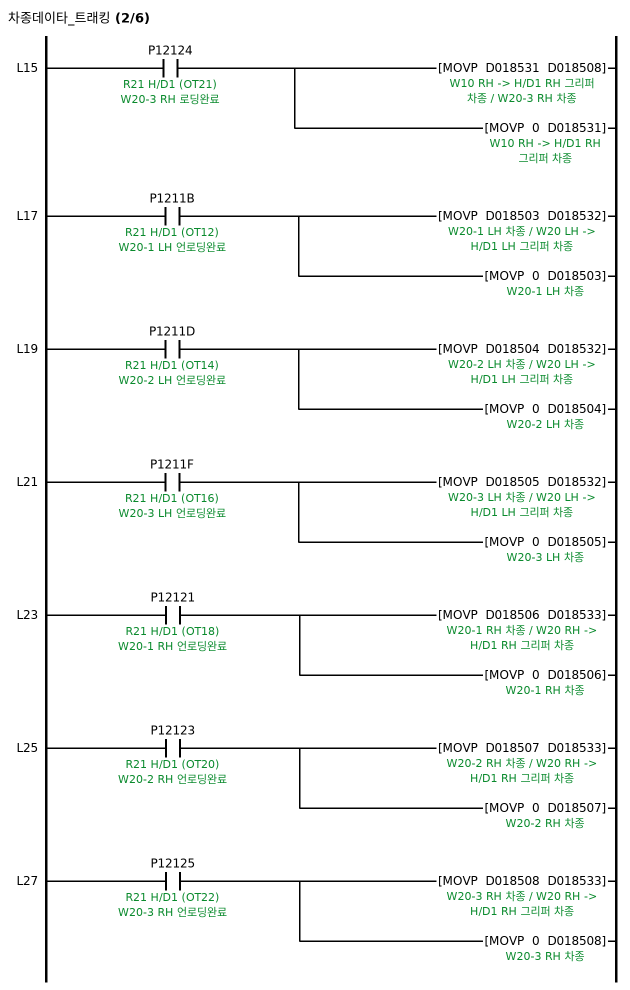
[picture p432: 차종데이타_트래킹 rungs L15-L27]
; L15
LOAD      P12124	// R21 H/D1 (OT21) W20-3 RH 로딩완료
MOVP      D018531 D018508	// W10 RH -> H/D1 RH 그리퍼 차종 / W20-3 RH 차종
MOVP      0 D018531	// W10 RH -> H/D1 RH 그리퍼 차종
; L17
LOAD      P1211B	// R21 H/D1 (OT12) W20-1 LH 언로딩완료
MOVP      D018503 D018532	// W20-1 LH 차종 / W20 LH -> H/D1 LH 그리퍼 차종
MOVP      0 D018503	// W20-1 LH 차종
; L19
LOAD      P1211D	// R21 H/D1 (OT14) W20-2 LH 언로딩완료
MOVP      D018504 D018532	// W20-2 LH 차종 / W20 LH -> H/D1 LH 그리퍼 차종
MOVP      0 D018504	// W20-2 LH 차종
; L21
LOAD      P1211F	// R21 H/D1 (OT16) W20-3 LH 언로딩완료
MOVP      D018505 D018532	// W20-3 LH 차종 / W20 LH -> H/D1 LH 그리퍼 차종
MOVP      0 D018505	// W20-3 LH 차종
; L23
LOAD      P12121	// R21 H/D1 (OT18) W20-1 RH 언로딩완료
MOVP      D018506 D018533	// W20-1 RH 차종 / W20 RH -> H/D1 RH 그리퍼 차종
MOVP      0 D018506	// W20-1 RH 차종
; L25
LOAD      P12123	// R21 H/D1 (OT20) W20-2 RH 언로딩완료
MOVP      D018507 D018533	// W20-2 RH 차종 / W20 RH -> H/D1 RH 그리퍼 차종
MOVP      0 D018507	// W20-2 RH 차종
; L27
LOAD      P12125	// R21 H/D1 (OT22) W20-3 RH 언로딩완료
MOVP      D018508 D018533	// W20-3 RH 차종 / W20 RH -> H/D1 RH 그리퍼 차종
MOVP      0 D018508	// W20-3 RH 차종

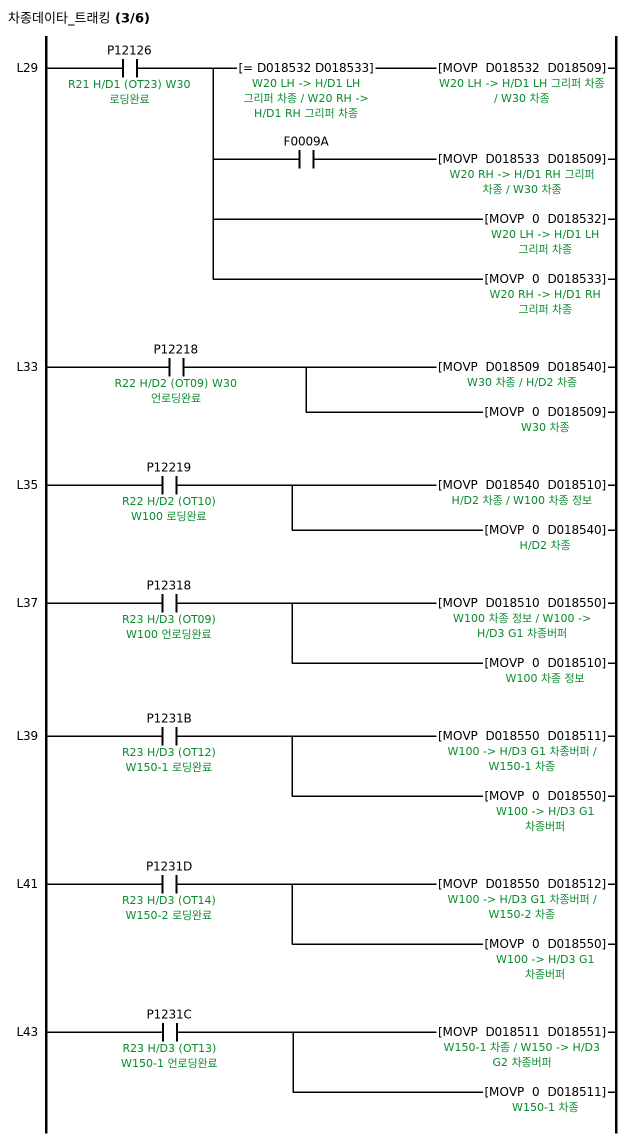
; L29
LOAD      P12126	// R21 H/D1 (OT23) W30 로딩완료
MPUSH
AND=      D018532 D018533	// W20 LH -> H/D1 LH 그리퍼 차종 / W20 RH -> H/D1 RH 그리퍼 차종
MOVP      D018532 D018509	// W20 LH -> H/D1 LH 그리퍼 차종 / W30 차종
MLOAD
AND       F0009A
MOVP      D018533 D018509	// W20 RH -> H/D1 RH 그리퍼 차종 / W30 차종
MPOP
MOVP      0 D018532	// W20 LH -> H/D1 LH 그리퍼 차종
MOVP      0 D018533	// W20 RH -> H/D1 RH 그리퍼 차종
; L33
LOAD      P12218	// R22 H/D2 (OT09) W30 언로딩완료
MOVP      D018509 D018540	// W30 차종 / H/D2 차종
MOVP      0 D018509	// W30 차종
; L35
LOAD      P12219	// R22 H/D2 (OT10) W100 로딩완료
MOVP      D018540 D018510	// H/D2 차종 / W100 차종 정보
MOVP      0 D018540	// H/D2 차종
; L37
LOAD      P12318	// R23 H/D3 (OT09) W100 언로딩완료
MOVP      D018510 D018550	// W100 차종 정보 / W100 -> H/D3 G1 차종버퍼
MOVP      0 D018510	// W100 차종 정보
; L39
LOAD      P1231B	// R23 H/D3 (OT12) W150-1 로딩완료
MOVP      D018550 D018511	// W100 -> H/D3 G1 차종버퍼 / W150-1 차종
MOVP      0 D018550	// W100 -> H/D3 G1 차종버퍼
; L41
LOAD      P1231D	// R23 H/D3 (OT14) W150-2 로딩완료
MOVP      D018550 D018512	// W100 -> H/D3 G1 차종버퍼 / W150-2 차종
MOVP      0 D018550	// W100 -> H/D3 G1 차종버퍼
; L43
LOAD      P1231C	// R23 H/D3 (OT13) W150-1 언로딩완료
MOVP      D018511 D018551	// W150-1 차종 / W150 -> H/D3 G2 차종버퍼
MOVP      0 D018511	// W150-1 차종

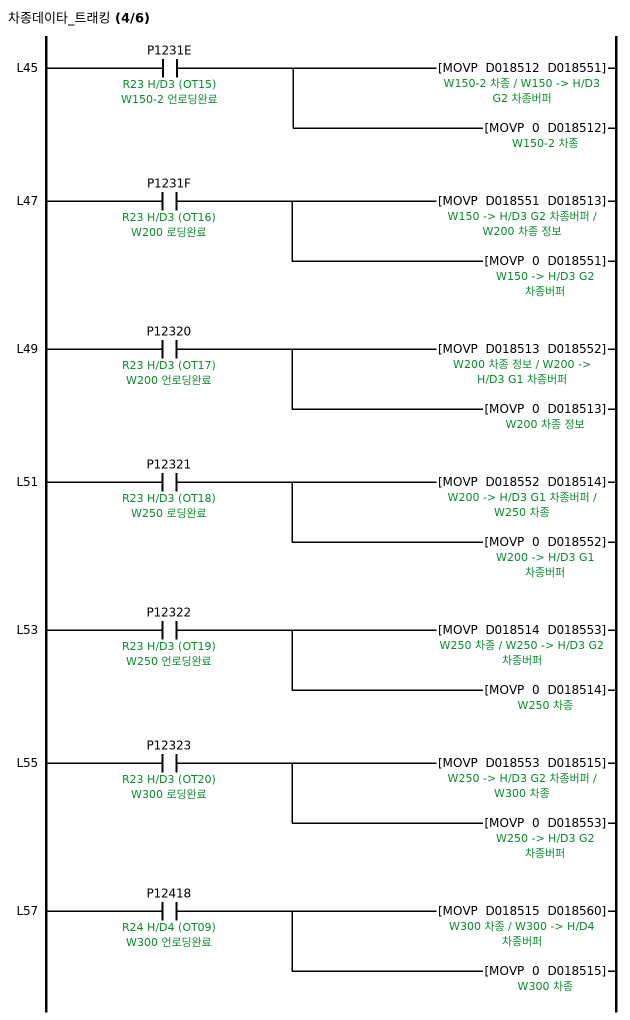
; L45
LOAD      P1231E	// R23 H/D3 (OT15) W150-2 언로딩완료
MOVP      D018512 D018551	// W150-2 차종 / W150 -> H/D3 G2 차종버퍼
MOVP      0 D018512	// W150-2 차종
; L47
LOAD      P1231F	// R23 H/D3 (OT16) W200 로딩완료
MOVP      D018551 D018513	// W150 -> H/D3 G2 차종버퍼 / W200 차종 정보
MOVP      0 D018551	// W150 -> H/D3 G2 차종버퍼
; L49
LOAD      P12320	// R23 H/D3 (OT17) W200 언로딩완료
MOVP      D018513 D018552	// W200 차종 정보 / W200 -> H/D3 G1 차종버퍼
MOVP      0 D018513	// W200 차종 정보
; L51
LOAD      P12321	// R23 H/D3 (OT18) W250 로딩완료
MOVP      D018552 D018514	// W200 -> H/D3 G1 차종버퍼 / W250 차종
MOVP      0 D018552	// W200 -> H/D3 G1 차종버퍼
; L53
LOAD      P12322	// R23 H/D3 (OT19) W250 언로딩완료
MOVP      D018514 D018553	// W250 차종 / W250 -> H/D3 G2 차종버퍼
MOVP      0 D018514	// W250 차종
; L55
LOAD      P12323	// R23 H/D3 (OT20) W300 로딩완료
MOVP      D018553 D018515	// W250 -> H/D3 G2 차종버퍼 / W300 차종
MOVP      0 D018553	// W250 -> H/D3 G2 차종버퍼
; L57
LOAD      P12418	// R24 H/D4 (OT09) W300 언로딩완료
MOVP      D018515 D018560	// W300 차종 / W300 -> H/D4 차종버퍼
MOVP      0 D018515	// W300 차종

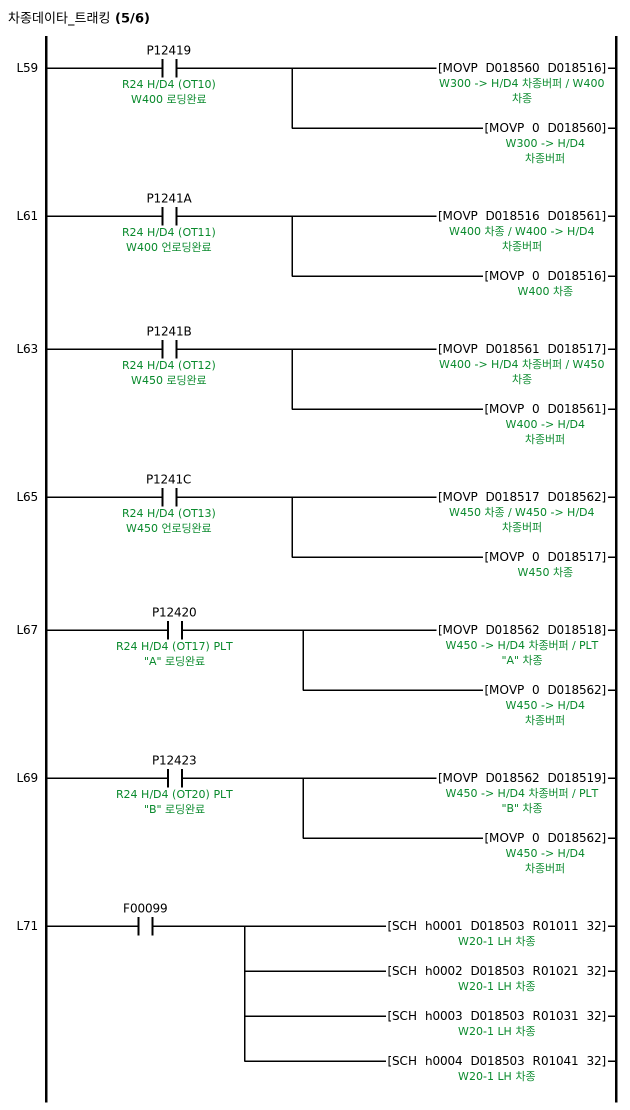
; L59
LOAD      P12419	// R24 H/D4 (OT10) W400 로딩완료
MOVP      D018560 D018516	// W300 -> H/D4 차종버퍼 / W400 차종
MOVP      0 D018560	// W300 -> H/D4 차종버퍼
; L61
LOAD      P1241A	// R24 H/D4 (OT11) W400 언로딩완료
MOVP      D018516 D018561	// W400 차종 / W400 -> H/D4 차종버퍼
MOVP      0 D018516	// W400 차종
; L63
LOAD      P1241B	// R24 H/D4 (OT12) W450 로딩완료
MOVP      D018561 D018517	// W400 -> H/D4 차종버퍼 / W450 차종
MOVP      0 D018561	// W400 -> H/D4 차종버퍼
; L65
LOAD      P1241C	// R24 H/D4 (OT13) W450 언로딩완료
MOVP      D018517 D018562	// W450 차종 / W450 -> H/D4 차종버퍼
MOVP      0 D018517	// W450 차종
; L67
LOAD      P12420	// R24 H/D4 (OT17) PLT "A" 로딩완료
MOVP      D018562 D018518	// W450 -> H/D4 차종버퍼 / PLT "A" 차종
MOVP      0 D018562	// W450 -> H/D4 차종버퍼
; L69
LOAD      P12423	// R24 H/D4 (OT20) PLT "B" 로딩완료
MOVP      D018562 D018519	// W450 -> H/D4 차종버퍼 / PLT "B" 차종
MOVP      0 D018562	// W450 -> H/D4 차종버퍼
; L71
LOAD      F00099
SCH       h0001 D018503 R01011 32	// W20-1 LH 차종
SCH       h0002 D018503 R01021 32	// W20-1 LH 차종
SCH       h0003 D018503 R01031 32	// W20-1 LH 차종
SCH       h0004 D018503 R01041 32	// W20-1 LH 차종

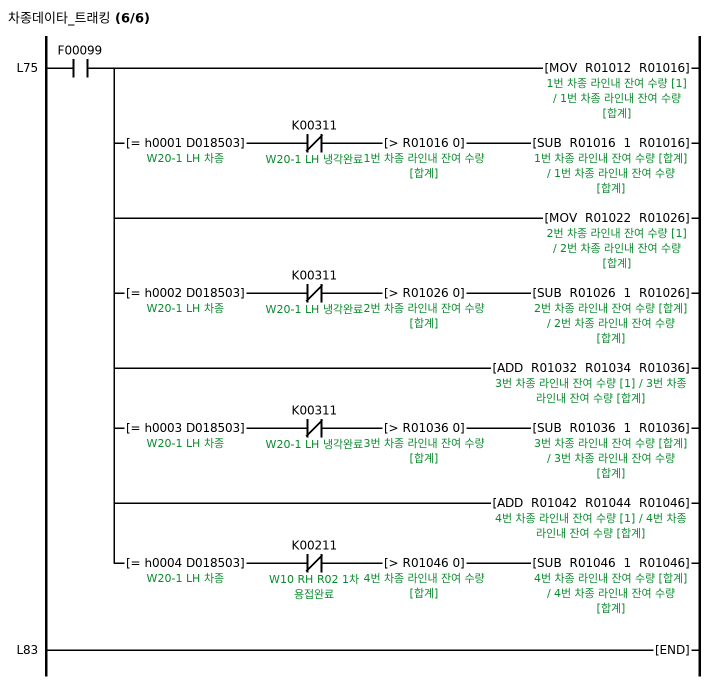
; L75
LOAD      F00099
MOV       R01012 R01016	// 1번 차종 라인내 잔여 수량 [1] / 1번 차종 라인내 잔여 수량 [합계]
MPUSH
AND=      h0001 D018503	// W20-1 LH 차종
AND NOT   K00311	// W20-1 LH 냉각완료
AND>      R01016 0	// 1번 차종 라인내 잔여 수량 [합계]
SUB       R01016 1 R01016	// 1번 차종 라인내 잔여 수량 [합계] / 1번 차종 라인내 잔여 수량 [합계]
MLOAD
MOV       R01022 R01026	// 2번 차종 라인내 잔여 수량 [1] / 2번 차종 라인내 잔여 수량 [합계]
AND=      h0002 D018503	// W20-1 LH 차종
AND NOT   K00311	// W20-1 LH 냉각완료
AND>      R01026 0	// 2번 차종 라인내 잔여 수량 [합계]
SUB       R01026 1 R01026	// 2번 차종 라인내 잔여 수량 [합계] / 2번 차종 라인내 잔여 수량 [합계]
MLOAD
ADD       R01032 R01034 R01036	// 3번 차종 라인내 잔여 수량 [1] / 3번 차종 라인내 잔여 수량 [합계]
AND=      h0003 D018503	// W20-1 LH 차종
AND NOT   K00311	// W20-1 LH 냉각완료
AND>      R01036 0	// 3번 차종 라인내 잔여 수량 [합계]
SUB       R01036 1 R01036	// 3번 차종 라인내 잔여 수량 [합계] / 3번 차종 라인내 잔여 수량 [합계]
MPOP
ADD       R01042 R01044 R01046	// 4번 차종 라인내 잔여 수량 [1] / 4번 차종 라인내 잔여 수량 [합계]
AND=      h0004 D018503	// W20-1 LH 차종
AND NOT   K00211	// W10 RH R02 1차 용접완료
AND>      R01046 0	// 4번 차종 라인내 잔여 수량 [합계]
SUB       R01046 1 R01046	// 4번 차종 라인내 잔여 수량 [합계] / 4번 차종 라인내 잔여 수량 [합계]
; L83
END

PROGRAM 마킹_지그데이타_트래킹 (task: 스캔 프로그램)

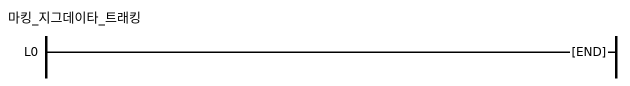
; L0
END

PROGRAM Car_Type (task: 스캔 프로그램)

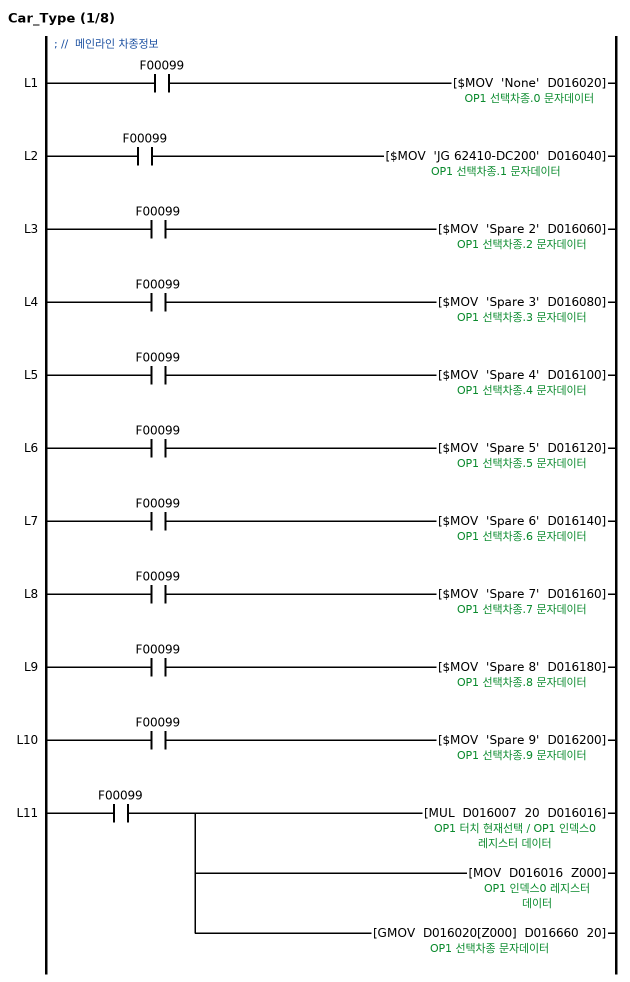
//   //  메인라인 차종정보
; L1
LOAD      F00099
$MOV      'None' D016020	// OP1 선택차종.0 문자데이터
; L2
LOAD      F00099
$MOV      'JG 62410-DC200' D016040	// OP1 선택차종.1 문자데이터
; L3
LOAD      F00099
$MOV      'Spare 2' D016060	// OP1 선택차종.2 문자데이터
; L4
LOAD      F00099
$MOV      'Spare 3' D016080	// OP1 선택차종.3 문자데이터
; L5
LOAD      F00099
$MOV      'Spare 4' D016100	// OP1 선택차종.4 문자데이터
; L6
LOAD      F00099
$MOV      'Spare 5' D016120	// OP1 선택차종.5 문자데이터
; L7
LOAD      F00099
$MOV      'Spare 6' D016140	// OP1 선택차종.6 문자데이터
; L8
LOAD      F00099
$MOV      'Spare 7' D016160	// OP1 선택차종.7 문자데이터
; L9
LOAD      F00099
$MOV      'Spare 8' D016180	// OP1 선택차종.8 문자데이터
; L10
LOAD      F00099
$MOV      'Spare 9' D016200	// OP1 선택차종.9 문자데이터
; L11
LOAD      F00099
MUL       D016007 20 D016016	// OP1 터치 현재선택 / OP1 인덱스0 레지스터 데이터
MOV       D016016 Z000	// OP1 인덱스0 레지스터 데이터
GMOV      D016020[Z000] D016660 20	// OP1 선택차종 문자데이터

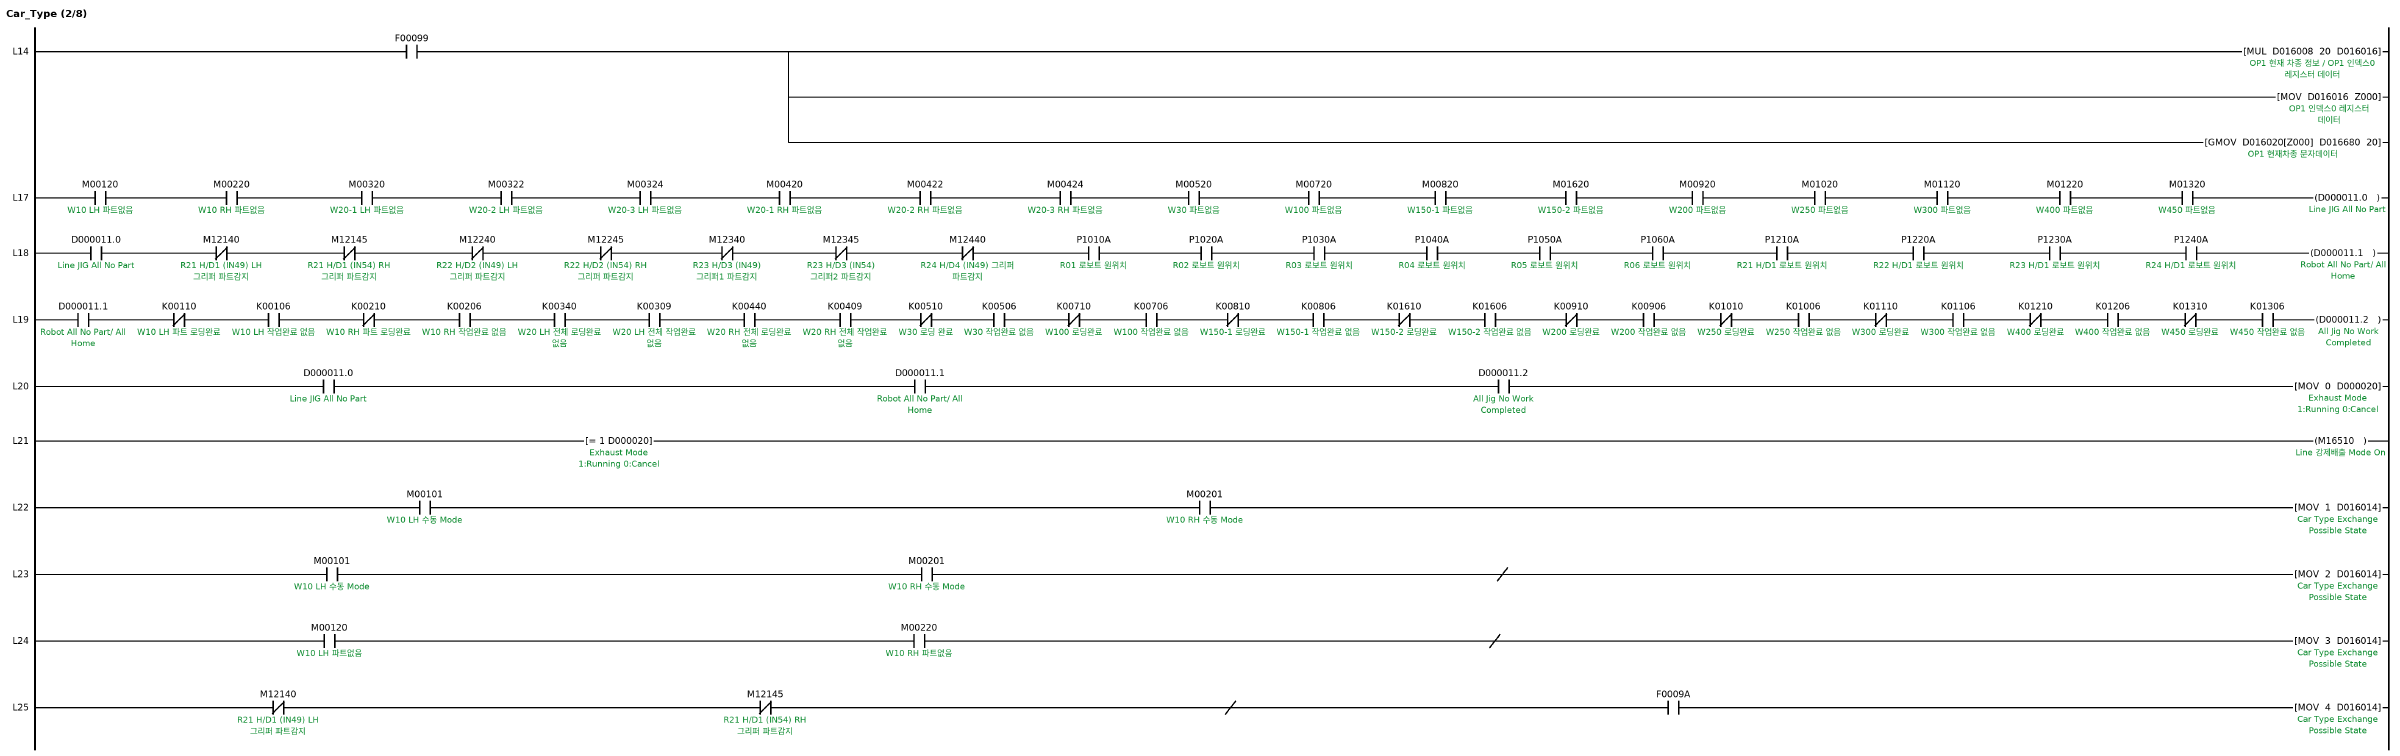
; L14
LOAD      F00099
MUL       D016008 20 D016016	// OP1 현재 차종 정보 / OP1 인덱스0 레지스터 데이터
MOV       D016016 Z000	// OP1 인덱스0 레지스터 데이터
GMOV      D016020[Z000] D016680 20	// OP1 현재차종 문자데이터
; L17
LOAD      M00120	// W10 LH 파트없음
AND       M00220	// W10 RH 파트없음
AND       M00320	// W20-1 LH 파트없음
AND       M00322	// W20-2 LH 파트없음
AND       M00324	// W20-3 LH 파트없음
AND       M00420	// W20-1 RH 파트없음
AND       M00422	// W20-2 RH 파트없음
AND       M00424	// W20-3 RH 파트없음
AND       M00520	// W30 파트없음
AND       M00720	// W100 파트없음
AND       M00820	// W150-1 파트없음
AND       M01620	// W150-2 파트없음
AND       M00920	// W200 파트없음
AND       M01020	// W250 파트없음
AND       M01120	// W300 파트없음
AND       M01220	// W400 파트없음
AND       M01320	// W450 파트없음
OUT       D000011.0	// Line JIG All No Part
; L18
LOAD      D000011.0	// Line JIG All No Part
AND NOT   M12140	// R21 H/D1 (IN49) LH 그리퍼 파트감지
AND NOT   M12145	// R21 H/D1 (IN54) RH 그리퍼 파트감지
AND NOT   M12240	// R22 H/D2 (IN49) LH 그리퍼 파트감지
AND NOT   M12245	// R22 H/D2 (IN54) RH 그리퍼 파트감지
AND NOT   M12340	// R23 H/D3 (IN49) 그리퍼1 파트감지
AND NOT   M12345	// R23 H/D3 (IN54) 그리퍼2 파트감지
AND NOT   M12440	// R24 H/D4 (IN49) 그리퍼 파트감지
AND       P1010A	// R01 로보트 원위치
AND       P1020A	// R02 로보트 원위치
AND       P1030A	// R03 로보트 원위치
AND       P1040A	// R04 로보트 원위치
AND       P1050A	// R05 로보트 원위치
AND       P1060A	// R06 로보트 원위치
AND       P1210A	// R21 H/D1 로보트 원위치
AND       P1220A	// R22 H/D1 로보트 원위치
AND       P1230A	// R23 H/D1 로보트 원위치
AND       P1240A	// R24 H/D1 로보트 원위치
OUT       D000011.1	// Robot All No Part/ All Home
; L19
LOAD      D000011.1	// Robot All No Part/ All Home
AND NOT   K00110	// W10 LH 파트 로딩완료
AND       K00106	// W10 LH 작업완료 없음
AND NOT   K00210	// W10 RH 파트 로딩완료
AND       K00206	// W10 RH 작업완료 없음
AND       K00340	// W20 LH 전체 로딩완료 없음
AND       K00309	// W20 LH 전체 작업완료 없음
AND       K00440	// W20 RH 전체 로딩완료 없음
AND       K00409	// W20 RH 전체 작업완료 없음
AND NOT   K00510	// W30 로딩 완료
AND       K00506	// W30 작업완료 없음
AND NOT   K00710	// W100 로딩완료
AND       K00706	// W100 작업완료 없음
AND NOT   K00810	// W150-1 로딩완료
AND       K00806	// W150-1 작업완료 없음
AND NOT   K01610	// W150-2 로딩완료
AND       K01606	// W150-2 작업완료 없음
AND NOT   K00910	// W200 로딩완료
AND       K00906	// W200 작업완료 없음
AND NOT   K01010	// W250 로딩완료
AND       K01006	// W250 작업완료 없음
AND NOT   K01110	// W300 로딩완료
AND       K01106	// W300 작업완료 없음
AND NOT   K01210	// W400 로딩완료
AND       K01206	// W400 작업완료 없음
AND NOT   K01310	// W450 로딩완료
AND       K01306	// W450 작업완료 없음
OUT       D000011.2	// All Jig No Work Completed
; L20
LOAD      D000011.0	// Line JIG All No Part
AND       D000011.1	// Robot All No Part/ All Home
AND       D000011.2	// All Jig No Work Completed
MOV       0 D000020	// Exhaust Mode 1:Running 0:Cancel
; L21
LOAD=     1 D000020	// Exhaust Mode 1:Running 0:Cancel
OUT       M16510	// Line 강제배출 Mode On
; L22
LOAD      M00101	// W10 LH 수동 Mode
AND       M00201	// W10 RH 수동 Mode
MOV       1 D016014	// Car Type Exchange Possible State
; L23
LOAD      M00101	// W10 LH 수동 Mode
AND       M00201	// W10 RH 수동 Mode
NOT
MOV       2 D016014	// Car Type Exchange Possible State
; L24
LOAD      M00120	// W10 LH 파트없음
AND       M00220	// W10 RH 파트없음
NOT
MOV       3 D016014	// Car Type Exchange Possible State
; L25
LOAD NOT  M12140	// R21 H/D1 (IN49) LH 그리퍼 파트감지
AND NOT   M12145	// R21 H/D1 (IN54) RH 그리퍼 파트감지
NOT
AND       F0009A
MOV       4 D016014	// Car Type Exchange Possible State

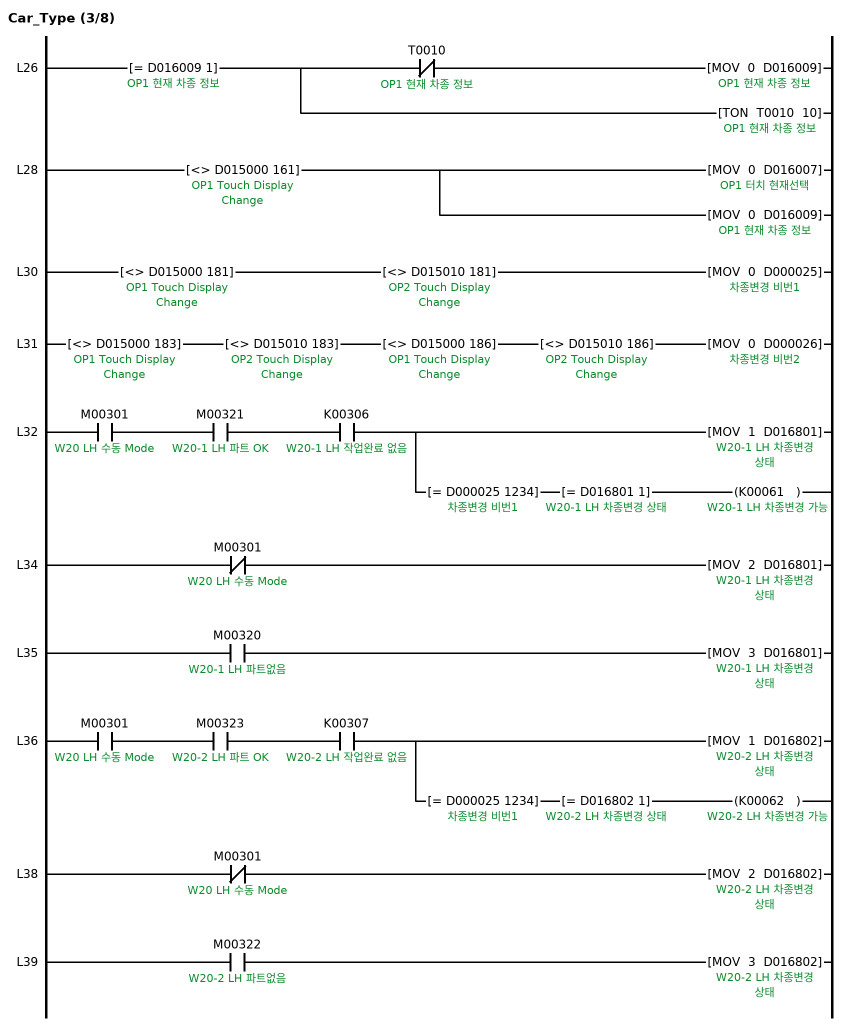
; L26
LOAD=     D016009 1	// OP1 현재 차종 정보
MPUSH
AND NOT   T0010	// OP1 현재 차종 정보
MOV       0 D016009	// OP1 현재 차종 정보
MPOP
TON       T0010 10	// OP1 현재 차종 정보
; L28
LOAD<>    D015000 161	// OP1 Touch Display Change
MOV       0 D016007	// OP1 터치 현재선택
MOV       0 D016009	// OP1 현재 차종 정보
; L30
LOAD<>    D015000 181	// OP1 Touch Display Change
AND<>     D015010 181	// OP2 Touch Display Change
MOV       0 D000025	// 차종변경 비번1
; L31
LOAD<>    D015000 183	// OP1 Touch Display Change
AND<>     D015010 183	// OP2 Touch Display Change
AND<>     D015000 186	// OP1 Touch Display Change
AND<>     D015010 186	// OP2 Touch Display Change
MOV       0 D000026	// 차종변경 비번2
; L32
LOAD      M00301	// W20 LH 수동 Mode
AND       M00321	// W20-1 LH 파트 OK
AND       K00306	// W20-1 LH 작업완료 없음
MOV       1 D016801	// W20-1 LH 차종변경 상태
AND=      D000025 1234	// 차종변경 비번1
AND=      D016801 1	// W20-1 LH 차종변경 상태
OUT       K00061	// W20-1 LH 차종변경 가능
; L34
LOAD NOT  M00301	// W20 LH 수동 Mode
MOV       2 D016801	// W20-1 LH 차종변경 상태
; L35
LOAD      M00320	// W20-1 LH 파트없음
MOV       3 D016801	// W20-1 LH 차종변경 상태
; L36
LOAD      M00301	// W20 LH 수동 Mode
AND       M00323	// W20-2 LH 파트 OK
AND       K00307	// W20-2 LH 작업완료 없음
MOV       1 D016802	// W20-2 LH 차종변경 상태
AND=      D000025 1234	// 차종변경 비번1
AND=      D016802 1	// W20-2 LH 차종변경 상태
OUT       K00062	// W20-2 LH 차종변경 가능
; L38
LOAD NOT  M00301	// W20 LH 수동 Mode
MOV       2 D016802	// W20-2 LH 차종변경 상태
; L39
LOAD      M00322	// W20-2 LH 파트없음
MOV       3 D016802	// W20-2 LH 차종변경 상태

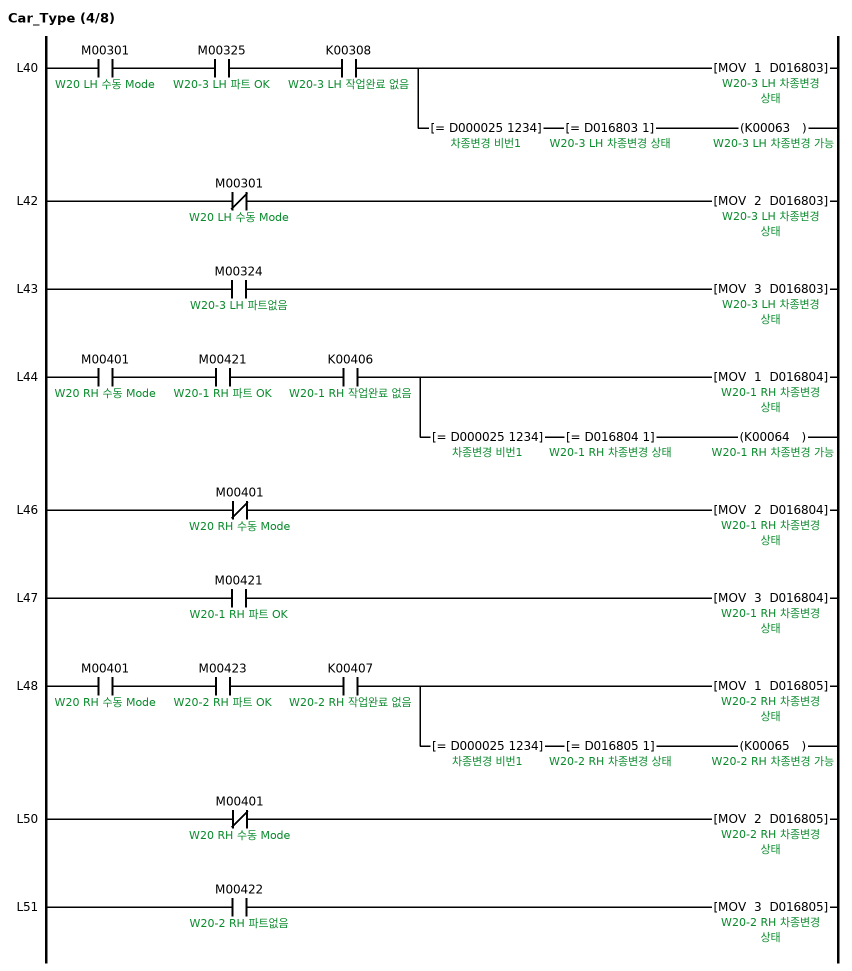
; L40
LOAD      M00301	// W20 LH 수동 Mode
AND       M00325	// W20-3 LH 파트 OK
AND       K00308	// W20-3 LH 작업완료 없음
MOV       1 D016803	// W20-3 LH 차종변경 상태
AND=      D000025 1234	// 차종변경 비번1
AND=      D016803 1	// W20-3 LH 차종변경 상태
OUT       K00063	// W20-3 LH 차종변경 가능
; L42
LOAD NOT  M00301	// W20 LH 수동 Mode
MOV       2 D016803	// W20-3 LH 차종변경 상태
; L43
LOAD      M00324	// W20-3 LH 파트없음
MOV       3 D016803	// W20-3 LH 차종변경 상태
; L44
LOAD      M00401	// W20 RH 수동 Mode
AND       M00421	// W20-1 RH 파트 OK
AND       K00406	// W20-1 RH 작업완료 없음
MOV       1 D016804	// W20-1 RH 차종변경 상태
AND=      D000025 1234	// 차종변경 비번1
AND=      D016804 1	// W20-1 RH 차종변경 상태
OUT       K00064	// W20-1 RH 차종변경 가능
; L46
LOAD NOT  M00401	// W20 RH 수동 Mode
MOV       2 D016804	// W20-1 RH 차종변경 상태
; L47
LOAD      M00421	// W20-1 RH 파트 OK
MOV       3 D016804	// W20-1 RH 차종변경 상태
; L48
LOAD      M00401	// W20 RH 수동 Mode
AND       M00423	// W20-2 RH 파트 OK
AND       K00407	// W20-2 RH 작업완료 없음
MOV       1 D016805	// W20-2 RH 차종변경 상태
AND=      D000025 1234	// 차종변경 비번1
AND=      D016805 1	// W20-2 RH 차종변경 상태
OUT       K00065	// W20-2 RH 차종변경 가능
; L50
LOAD NOT  M00401	// W20 RH 수동 Mode
MOV       2 D016805	// W20-2 RH 차종변경 상태
; L51
LOAD      M00422	// W20-2 RH 파트없음
MOV       3 D016805	// W20-2 RH 차종변경 상태

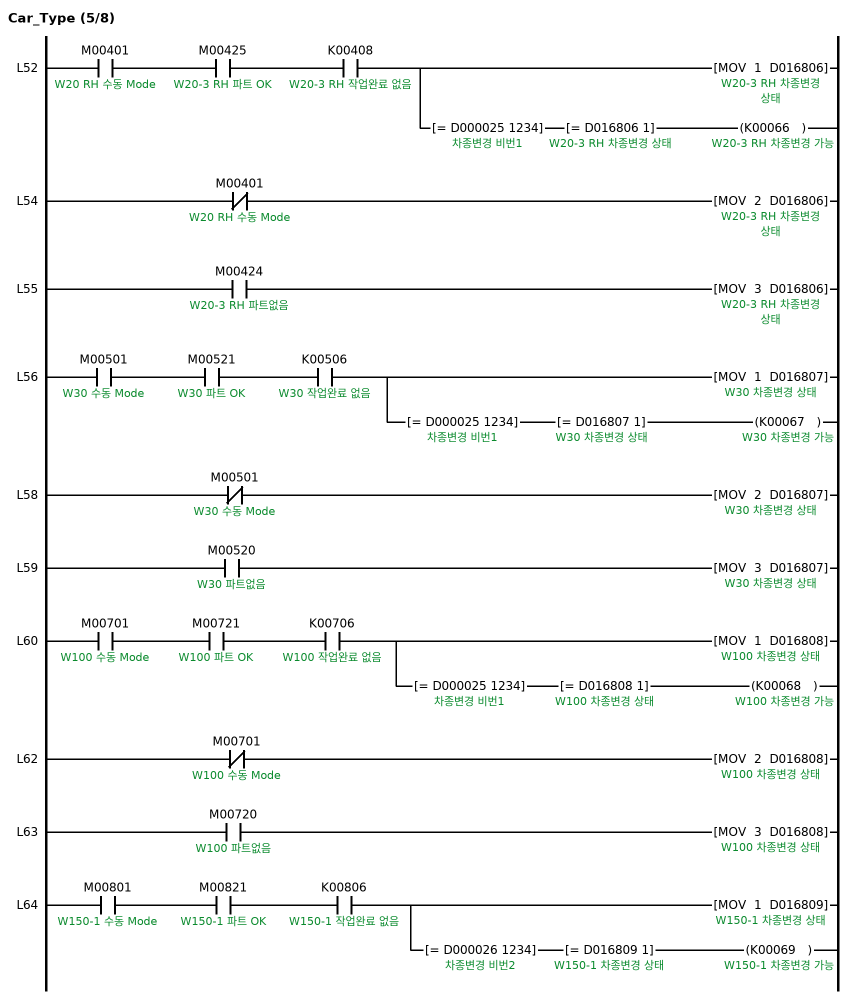
; L52
LOAD      M00401	// W20 RH 수동 Mode
AND       M00425	// W20-3 RH 파트 OK
AND       K00408	// W20-3 RH 작업완료 없음
MOV       1 D016806	// W20-3 RH 차종변경 상태
AND=      D000025 1234	// 차종변경 비번1
AND=      D016806 1	// W20-3 RH 차종변경 상태
OUT       K00066	// W20-3 RH 차종변경 가능
; L54
LOAD NOT  M00401	// W20 RH 수동 Mode
MOV       2 D016806	// W20-3 RH 차종변경 상태
; L55
LOAD      M00424	// W20-3 RH 파트없음
MOV       3 D016806	// W20-3 RH 차종변경 상태
; L56
LOAD      M00501	// W30 수동 Mode
AND       M00521	// W30 파트 OK
AND       K00506	// W30 작업완료 없음
MOV       1 D016807	// W30 차종변경 상태
AND=      D000025 1234	// 차종변경 비번1
AND=      D016807 1	// W30 차종변경 상태
OUT       K00067	// W30 차종변경 가능
; L58
LOAD NOT  M00501	// W30 수동 Mode
MOV       2 D016807	// W30 차종변경 상태
; L59
LOAD      M00520	// W30 파트없음
MOV       3 D016807	// W30 차종변경 상태
; L60
LOAD      M00701	// W100 수동 Mode
AND       M00721	// W100 파트 OK
AND       K00706	// W100 작업완료 없음
MOV       1 D016808	// W100 차종변경 상태
AND=      D000025 1234	// 차종변경 비번1
AND=      D016808 1	// W100 차종변경 상태
OUT       K00068	// W100 차종변경 가능
; L62
LOAD NOT  M00701	// W100 수동 Mode
MOV       2 D016808	// W100 차종변경 상태
; L63
LOAD      M00720	// W100 파트없음
MOV       3 D016808	// W100 차종변경 상태
; L64
LOAD      M00801	// W150-1 수동 Mode
AND       M00821	// W150-1 파트 OK
AND       K00806	// W150-1 작업완료 없음
MOV       1 D016809	// W150-1 차종변경 상태
AND=      D000026 1234	// 차종변경 비번2
AND=      D016809 1	// W150-1 차종변경 상태
OUT       K00069	// W150-1 차종변경 가능

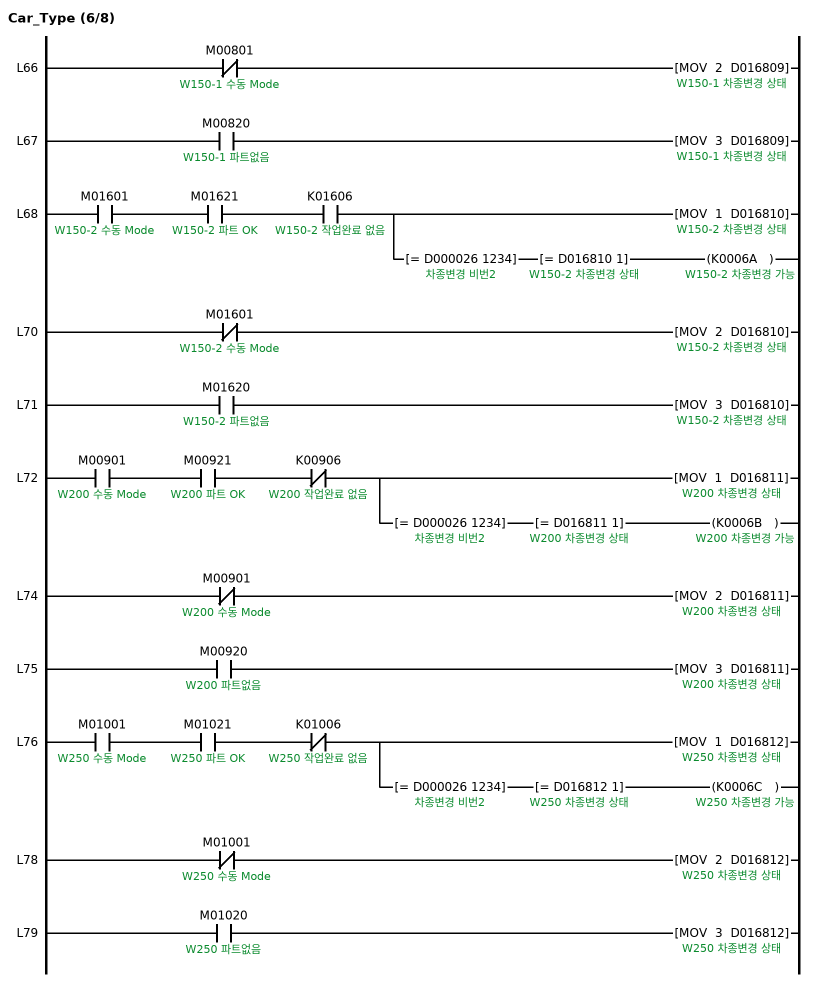
; L66
LOAD NOT  M00801	// W150-1 수동 Mode
MOV       2 D016809	// W150-1 차종변경 상태
; L67
LOAD      M00820	// W150-1 파트없음
MOV       3 D016809	// W150-1 차종변경 상태
; L68
LOAD      M01601	// W150-2 수동 Mode
AND       M01621	// W150-2 파트 OK
AND       K01606	// W150-2 작업완료 없음
MOV       1 D016810	// W150-2 차종변경 상태
AND=      D000026 1234	// 차종변경 비번2
AND=      D016810 1	// W150-2 차종변경 상태
OUT       K0006A	// W150-2 차종변경 가능
; L70
LOAD NOT  M01601	// W150-2 수동 Mode
MOV       2 D016810	// W150-2 차종변경 상태
; L71
LOAD      M01620	// W150-2 파트없음
MOV       3 D016810	// W150-2 차종변경 상태
; L72
LOAD      M00901	// W200 수동 Mode
AND       M00921	// W200 파트 OK
AND NOT   K00906	// W200 작업완료 없음
MOV       1 D016811	// W200 차종변경 상태
AND=      D000026 1234	// 차종변경 비번2
AND=      D016811 1	// W200 차종변경 상태
OUT       K0006B	// W200 차종변경 가능
; L74
LOAD NOT  M00901	// W200 수동 Mode
MOV       2 D016811	// W200 차종변경 상태
; L75
LOAD      M00920	// W200 파트없음
MOV       3 D016811	// W200 차종변경 상태
; L76
LOAD      M01001	// W250 수동 Mode
AND       M01021	// W250 파트 OK
AND NOT   K01006	// W250 작업완료 없음
MOV       1 D016812	// W250 차종변경 상태
AND=      D000026 1234	// 차종변경 비번2
AND=      D016812 1	// W250 차종변경 상태
OUT       K0006C	// W250 차종변경 가능
; L78
LOAD NOT  M01001	// W250 수동 Mode
MOV       2 D016812	// W250 차종변경 상태
; L79
LOAD      M01020	// W250 파트없음
MOV       3 D016812	// W250 차종변경 상태

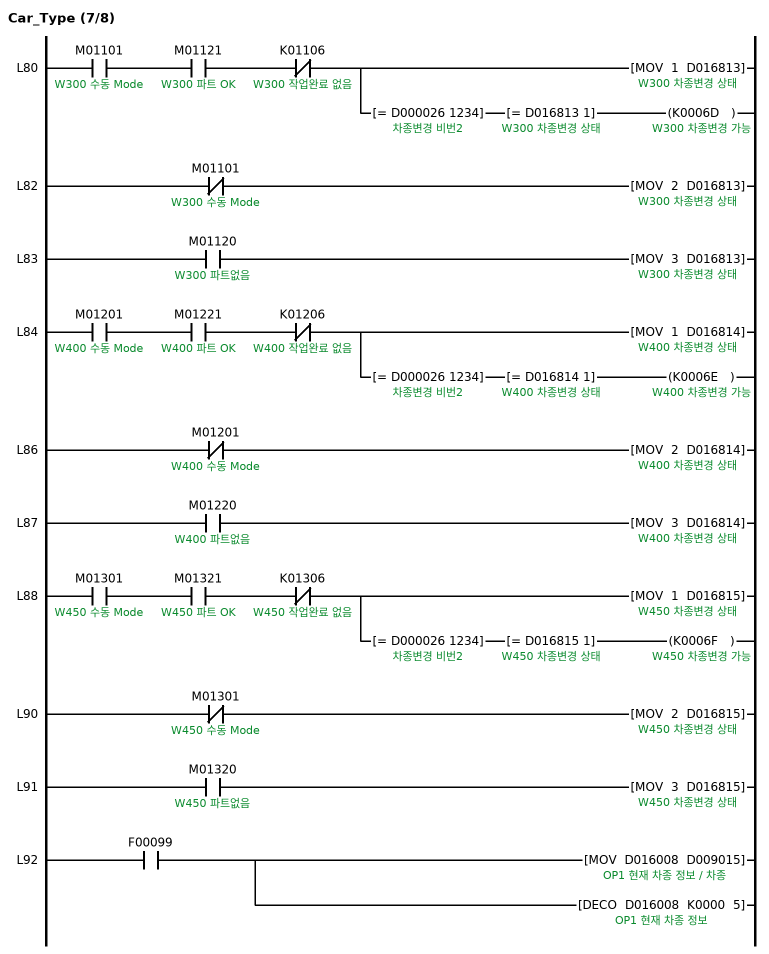
; L80
LOAD      M01101	// W300 수동 Mode
AND       M01121	// W300 파트 OK
AND NOT   K01106	// W300 작업완료 없음
MOV       1 D016813	// W300 차종변경 상태
AND=      D000026 1234	// 차종변경 비번2
AND=      D016813 1	// W300 차종변경 상태
OUT       K0006D	// W300 차종변경 가능
; L82
LOAD NOT  M01101	// W300 수동 Mode
MOV       2 D016813	// W300 차종변경 상태
; L83
LOAD      M01120	// W300 파트없음
MOV       3 D016813	// W300 차종변경 상태
; L84
LOAD      M01201	// W400 수동 Mode
AND       M01221	// W400 파트 OK
AND NOT   K01206	// W400 작업완료 없음
MOV       1 D016814	// W400 차종변경 상태
AND=      D000026 1234	// 차종변경 비번2
AND=      D016814 1	// W400 차종변경 상태
OUT       K0006E	// W400 차종변경 가능
; L86
LOAD NOT  M01201	// W400 수동 Mode
MOV       2 D016814	// W400 차종변경 상태
; L87
LOAD      M01220	// W400 파트없음
MOV       3 D016814	// W400 차종변경 상태
; L88
LOAD      M01301	// W450 수동 Mode
AND       M01321	// W450 파트 OK
AND NOT   K01306	// W450 작업완료 없음
MOV       1 D016815	// W450 차종변경 상태
AND=      D000026 1234	// 차종변경 비번2
AND=      D016815 1	// W450 차종변경 상태
OUT       K0006F	// W450 차종변경 가능
; L90
LOAD NOT  M01301	// W450 수동 Mode
MOV       2 D016815	// W450 차종변경 상태
; L91
LOAD      M01320	// W450 파트없음
MOV       3 D016815	// W450 차종변경 상태
; L92
LOAD      F00099
MOV       D016008 D009015	// OP1 현재 차종 정보 / 차종
DECO      D016008 K0000 5	// OP1 현재 차종 정보

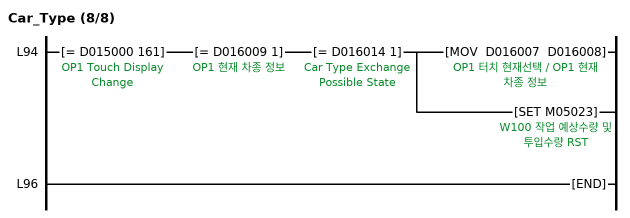
; L94
LOAD=     D015000 161	// OP1 Touch Display Change
AND=      D016009 1	// OP1 현재 차종 정보
AND=      D016014 1	// Car Type Exchange Possible State
MOV       D016007 D016008	// OP1 터치 현재선택 / OP1 현재 차종 정보
SET       M05023	// W100 작업 예상수량 및 투입수량 RST
; L96
END

PROGRAM 생산관리 (task: 스캔 프로그램)

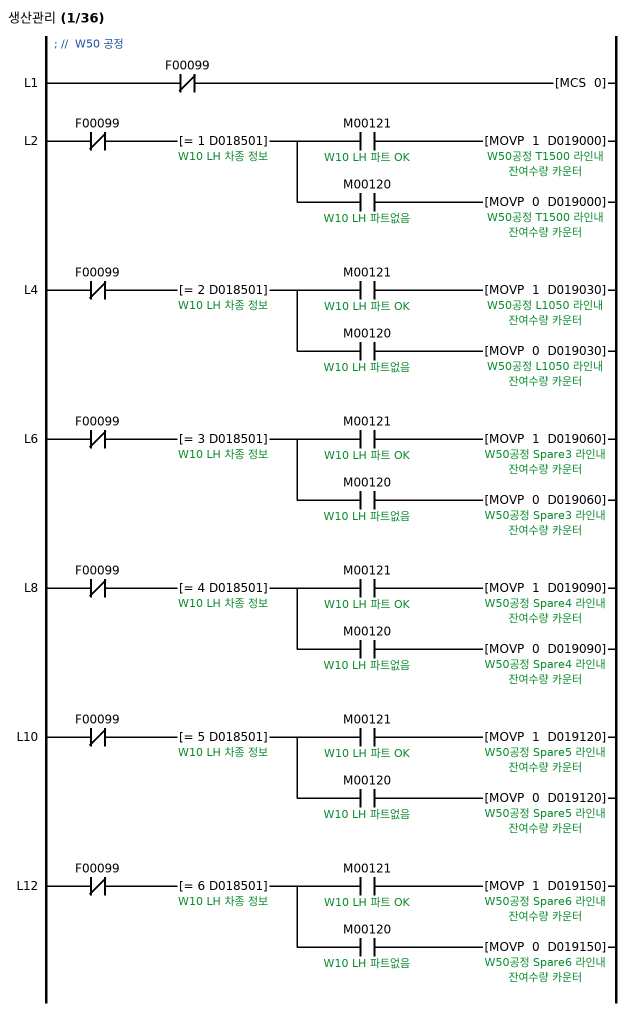
//   //  W50 공정
; L1
LOAD NOT  F00099
MCS       0
; L2
LOAD NOT  F00099
AND=      1 D018501	// W10 LH 차종 정보
MPUSH
AND       M00121	// W10 LH 파트 OK
MOVP      1 D019000	// W50공정 T1500 라인내 잔여수량 카운터
MPOP
AND       M00120	// W10 LH 파트없음
MOVP      0 D019000	// W50공정 T1500 라인내 잔여수량 카운터
; L4
LOAD NOT  F00099
AND=      2 D018501	// W10 LH 차종 정보
MPUSH
AND       M00121	// W10 LH 파트 OK
MOVP      1 D019030	// W50공정 L1050 라인내 잔여수량 카운터
MPOP
AND       M00120	// W10 LH 파트없음
MOVP      0 D019030	// W50공정 L1050 라인내 잔여수량 카운터
; L6
LOAD NOT  F00099
AND=      3 D018501	// W10 LH 차종 정보
MPUSH
AND       M00121	// W10 LH 파트 OK
MOVP      1 D019060	// W50공정 Spare3 라인내 잔여수량 카운터
MPOP
AND       M00120	// W10 LH 파트없음
MOVP      0 D019060	// W50공정 Spare3 라인내 잔여수량 카운터
; L8
LOAD NOT  F00099
AND=      4 D018501	// W10 LH 차종 정보
MPUSH
AND       M00121	// W10 LH 파트 OK
MOVP      1 D019090	// W50공정 Spare4 라인내 잔여수량 카운터
MPOP
AND       M00120	// W10 LH 파트없음
MOVP      0 D019090	// W50공정 Spare4 라인내 잔여수량 카운터
; L10
LOAD NOT  F00099
AND=      5 D018501	// W10 LH 차종 정보
MPUSH
AND       M00121	// W10 LH 파트 OK
MOVP      1 D019120	// W50공정 Spare5 라인내 잔여수량 카운터
MPOP
AND       M00120	// W10 LH 파트없음
MOVP      0 D019120	// W50공정 Spare5 라인내 잔여수량 카운터
; L12
LOAD NOT  F00099
AND=      6 D018501	// W10 LH 차종 정보
MPUSH
AND       M00121	// W10 LH 파트 OK
MOVP      1 D019150	// W50공정 Spare6 라인내 잔여수량 카운터
MPOP
AND       M00120	// W10 LH 파트없음
MOVP      0 D019150	// W50공정 Spare6 라인내 잔여수량 카운터

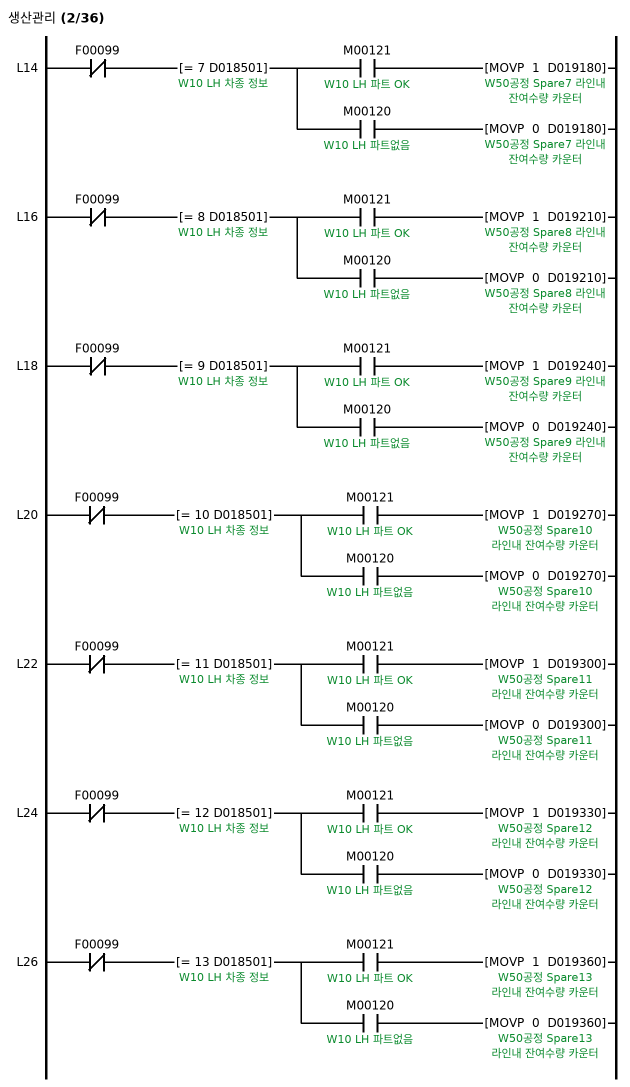
; L14
LOAD NOT  F00099
AND=      7 D018501	// W10 LH 차종 정보
MPUSH
AND       M00121	// W10 LH 파트 OK
MOVP      1 D019180	// W50공정 Spare7 라인내 잔여수량 카운터
MPOP
AND       M00120	// W10 LH 파트없음
MOVP      0 D019180	// W50공정 Spare7 라인내 잔여수량 카운터
; L16
LOAD NOT  F00099
AND=      8 D018501	// W10 LH 차종 정보
MPUSH
AND       M00121	// W10 LH 파트 OK
MOVP      1 D019210	// W50공정 Spare8 라인내 잔여수량 카운터
MPOP
AND       M00120	// W10 LH 파트없음
MOVP      0 D019210	// W50공정 Spare8 라인내 잔여수량 카운터
; L18
LOAD NOT  F00099
AND=      9 D018501	// W10 LH 차종 정보
MPUSH
AND       M00121	// W10 LH 파트 OK
MOVP      1 D019240	// W50공정 Spare9 라인내 잔여수량 카운터
MPOP
AND       M00120	// W10 LH 파트없음
MOVP      0 D019240	// W50공정 Spare9 라인내 잔여수량 카운터
; L20
LOAD NOT  F00099
AND=      10 D018501	// W10 LH 차종 정보
MPUSH
AND       M00121	// W10 LH 파트 OK
MOVP      1 D019270	// W50공정 Spare10 라인내 잔여수량 카운터
MPOP
AND       M00120	// W10 LH 파트없음
MOVP      0 D019270	// W50공정 Spare10 라인내 잔여수량 카운터
; L22
LOAD NOT  F00099
AND=      11 D018501	// W10 LH 차종 정보
MPUSH
AND       M00121	// W10 LH 파트 OK
MOVP      1 D019300	// W50공정 Spare11 라인내 잔여수량 카운터
MPOP
AND       M00120	// W10 LH 파트없음
MOVP      0 D019300	// W50공정 Spare11 라인내 잔여수량 카운터
; L24
LOAD NOT  F00099
AND=      12 D018501	// W10 LH 차종 정보
MPUSH
AND       M00121	// W10 LH 파트 OK
MOVP      1 D019330	// W50공정 Spare12 라인내 잔여수량 카운터
MPOP
AND       M00120	// W10 LH 파트없음
MOVP      0 D019330	// W50공정 Spare12 라인내 잔여수량 카운터
; L26
LOAD NOT  F00099
AND=      13 D018501	// W10 LH 차종 정보
MPUSH
AND       M00121	// W10 LH 파트 OK
MOVP      1 D019360	// W50공정 Spare13 라인내 잔여수량 카운터
MPOP
AND       M00120	// W10 LH 파트없음
MOVP      0 D019360	// W50공정 Spare13 라인내 잔여수량 카운터

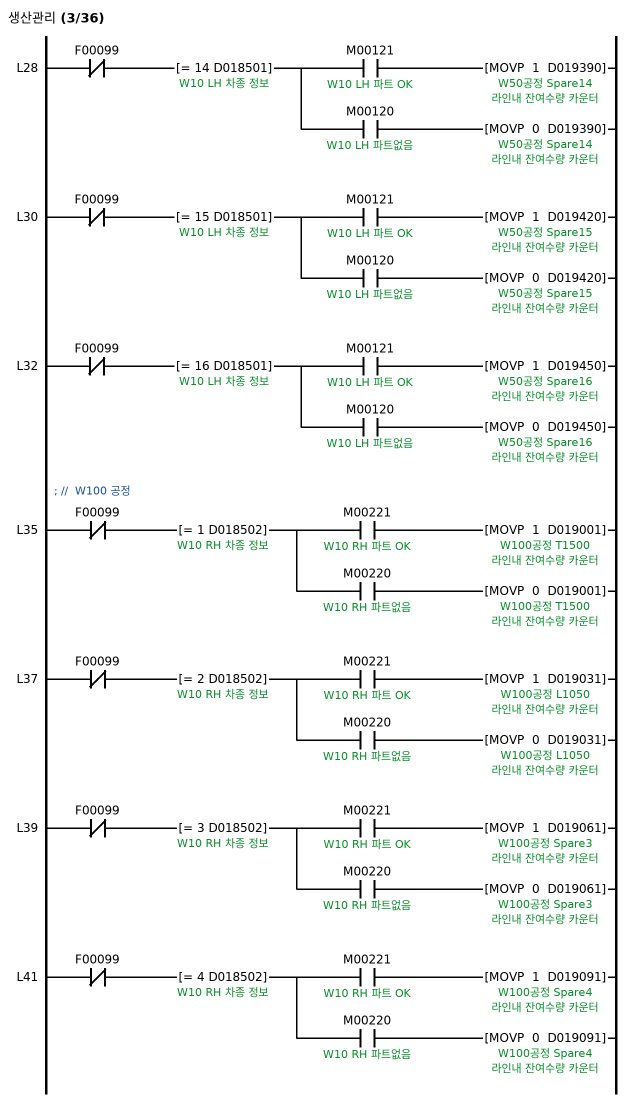
; L28
LOAD NOT  F00099
AND=      14 D018501	// W10 LH 차종 정보
MPUSH
AND       M00121	// W10 LH 파트 OK
MOVP      1 D019390	// W50공정 Spare14 라인내 잔여수량 카운터
MPOP
AND       M00120	// W10 LH 파트없음
MOVP      0 D019390	// W50공정 Spare14 라인내 잔여수량 카운터
; L30
LOAD NOT  F00099
AND=      15 D018501	// W10 LH 차종 정보
MPUSH
AND       M00121	// W10 LH 파트 OK
MOVP      1 D019420	// W50공정 Spare15 라인내 잔여수량 카운터
MPOP
AND       M00120	// W10 LH 파트없음
MOVP      0 D019420	// W50공정 Spare15 라인내 잔여수량 카운터
; L32
LOAD NOT  F00099
AND=      16 D018501	// W10 LH 차종 정보
MPUSH
AND       M00121	// W10 LH 파트 OK
MOVP      1 D019450	// W50공정 Spare16 라인내 잔여수량 카운터
MPOP
AND       M00120	// W10 LH 파트없음
MOVP      0 D019450	// W50공정 Spare16 라인내 잔여수량 카운터
//   //  W100 공정
; L35
LOAD NOT  F00099
AND=      1 D018502	// W10 RH 차종 정보
MPUSH
AND       M00221	// W10 RH 파트 OK
MOVP      1 D019001	// W100공정 T1500 라인내 잔여수량 카운터
MPOP
AND       M00220	// W10 RH 파트없음
MOVP      0 D019001	// W100공정 T1500 라인내 잔여수량 카운터
; L37
LOAD NOT  F00099
AND=      2 D018502	// W10 RH 차종 정보
MPUSH
AND       M00221	// W10 RH 파트 OK
MOVP      1 D019031	// W100공정 L1050 라인내 잔여수량 카운터
MPOP
AND       M00220	// W10 RH 파트없음
MOVP      0 D019031	// W100공정 L1050 라인내 잔여수량 카운터
; L39
LOAD NOT  F00099
AND=      3 D018502	// W10 RH 차종 정보
MPUSH
AND       M00221	// W10 RH 파트 OK
MOVP      1 D019061	// W100공정 Spare3 라인내 잔여수량 카운터
MPOP
AND       M00220	// W10 RH 파트없음
MOVP      0 D019061	// W100공정 Spare3 라인내 잔여수량 카운터
; L41
LOAD NOT  F00099
AND=      4 D018502	// W10 RH 차종 정보
MPUSH
AND       M00221	// W10 RH 파트 OK
MOVP      1 D019091	// W100공정 Spare4 라인내 잔여수량 카운터
MPOP
AND       M00220	// W10 RH 파트없음
MOVP      0 D019091	// W100공정 Spare4 라인내 잔여수량 카운터

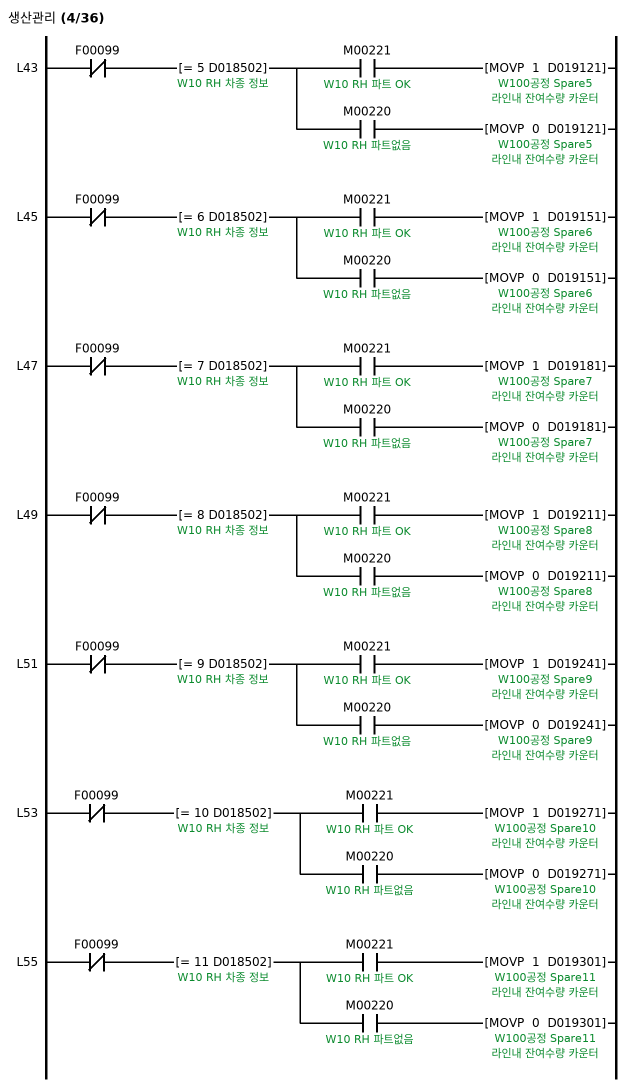
; L43
LOAD NOT  F00099
AND=      5 D018502	// W10 RH 차종 정보
MPUSH
AND       M00221	// W10 RH 파트 OK
MOVP      1 D019121	// W100공정 Spare5 라인내 잔여수량 카운터
MPOP
AND       M00220	// W10 RH 파트없음
MOVP      0 D019121	// W100공정 Spare5 라인내 잔여수량 카운터
; L45
LOAD NOT  F00099
AND=      6 D018502	// W10 RH 차종 정보
MPUSH
AND       M00221	// W10 RH 파트 OK
MOVP      1 D019151	// W100공정 Spare6 라인내 잔여수량 카운터
MPOP
AND       M00220	// W10 RH 파트없음
MOVP      0 D019151	// W100공정 Spare6 라인내 잔여수량 카운터
; L47
LOAD NOT  F00099
AND=      7 D018502	// W10 RH 차종 정보
MPUSH
AND       M00221	// W10 RH 파트 OK
MOVP      1 D019181	// W100공정 Spare7 라인내 잔여수량 카운터
MPOP
AND       M00220	// W10 RH 파트없음
MOVP      0 D019181	// W100공정 Spare7 라인내 잔여수량 카운터
; L49
LOAD NOT  F00099
AND=      8 D018502	// W10 RH 차종 정보
MPUSH
AND       M00221	// W10 RH 파트 OK
MOVP      1 D019211	// W100공정 Spare8 라인내 잔여수량 카운터
MPOP
AND       M00220	// W10 RH 파트없음
MOVP      0 D019211	// W100공정 Spare8 라인내 잔여수량 카운터
; L51
LOAD NOT  F00099
AND=      9 D018502	// W10 RH 차종 정보
MPUSH
AND       M00221	// W10 RH 파트 OK
MOVP      1 D019241	// W100공정 Spare9 라인내 잔여수량 카운터
MPOP
AND       M00220	// W10 RH 파트없음
MOVP      0 D019241	// W100공정 Spare9 라인내 잔여수량 카운터
; L53
LOAD NOT  F00099
AND=      10 D018502	// W10 RH 차종 정보
MPUSH
AND       M00221	// W10 RH 파트 OK
MOVP      1 D019271	// W100공정 Spare10 라인내 잔여수량 카운터
MPOP
AND       M00220	// W10 RH 파트없음
MOVP      0 D019271	// W100공정 Spare10 라인내 잔여수량 카운터
; L55
LOAD NOT  F00099
AND=      11 D018502	// W10 RH 차종 정보
MPUSH
AND       M00221	// W10 RH 파트 OK
MOVP      1 D019301	// W100공정 Spare11 라인내 잔여수량 카운터
MPOP
AND       M00220	// W10 RH 파트없음
MOVP      0 D019301	// W100공정 Spare11 라인내 잔여수량 카운터

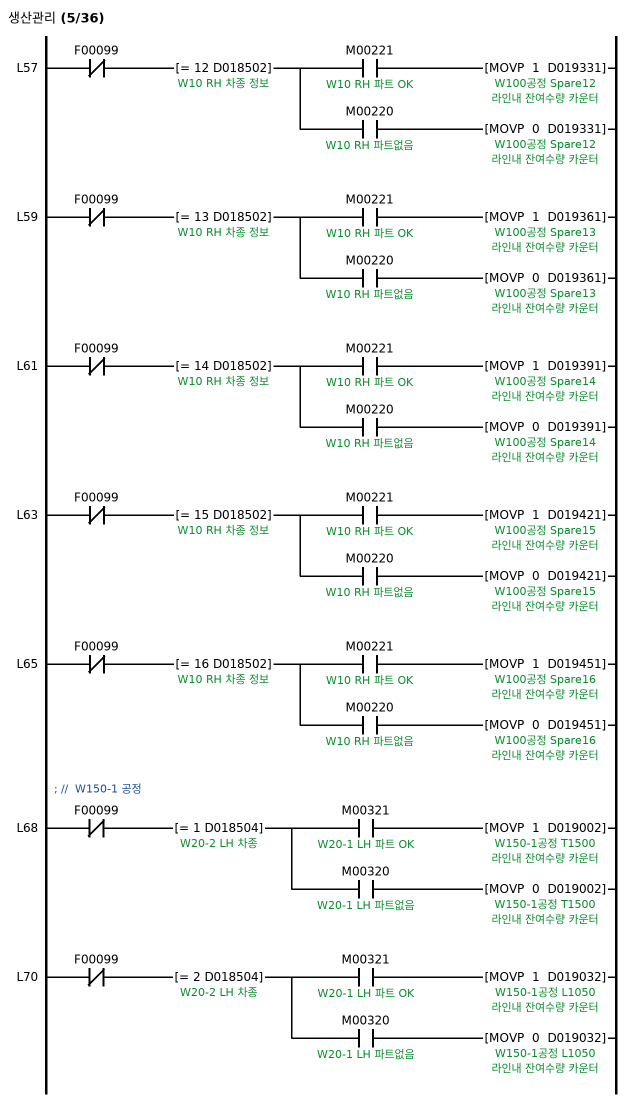
; L57
LOAD NOT  F00099
AND=      12 D018502	// W10 RH 차종 정보
MPUSH
AND       M00221	// W10 RH 파트 OK
MOVP      1 D019331	// W100공정 Spare12 라인내 잔여수량 카운터
MPOP
AND       M00220	// W10 RH 파트없음
MOVP      0 D019331	// W100공정 Spare12 라인내 잔여수량 카운터
; L59
LOAD NOT  F00099
AND=      13 D018502	// W10 RH 차종 정보
MPUSH
AND       M00221	// W10 RH 파트 OK
MOVP      1 D019361	// W100공정 Spare13 라인내 잔여수량 카운터
MPOP
AND       M00220	// W10 RH 파트없음
MOVP      0 D019361	// W100공정 Spare13 라인내 잔여수량 카운터
; L61
LOAD NOT  F00099
AND=      14 D018502	// W10 RH 차종 정보
MPUSH
AND       M00221	// W10 RH 파트 OK
MOVP      1 D019391	// W100공정 Spare14 라인내 잔여수량 카운터
MPOP
AND       M00220	// W10 RH 파트없음
MOVP      0 D019391	// W100공정 Spare14 라인내 잔여수량 카운터
; L63
LOAD NOT  F00099
AND=      15 D018502	// W10 RH 차종 정보
MPUSH
AND       M00221	// W10 RH 파트 OK
MOVP      1 D019421	// W100공정 Spare15 라인내 잔여수량 카운터
MPOP
AND       M00220	// W10 RH 파트없음
MOVP      0 D019421	// W100공정 Spare15 라인내 잔여수량 카운터
; L65
LOAD NOT  F00099
AND=      16 D018502	// W10 RH 차종 정보
MPUSH
AND       M00221	// W10 RH 파트 OK
MOVP      1 D019451	// W100공정 Spare16 라인내 잔여수량 카운터
MPOP
AND       M00220	// W10 RH 파트없음
MOVP      0 D019451	// W100공정 Spare16 라인내 잔여수량 카운터
//   //  W150-1 공정
; L68
LOAD NOT  F00099
AND=      1 D018504	// W20-2 LH 차종
MPUSH
AND       M00321	// W20-1 LH 파트 OK
MOVP      1 D019002	// W150-1공정 T1500 라인내 잔여수량 카운터
MPOP
AND       M00320	// W20-1 LH 파트없음
MOVP      0 D019002	// W150-1공정 T1500 라인내 잔여수량 카운터
; L70
LOAD NOT  F00099
AND=      2 D018504	// W20-2 LH 차종
MPUSH
AND       M00321	// W20-1 LH 파트 OK
MOVP      1 D019032	// W150-1공정 L1050 라인내 잔여수량 카운터
MPOP
AND       M00320	// W20-1 LH 파트없음
MOVP      0 D019032	// W150-1공정 L1050 라인내 잔여수량 카운터

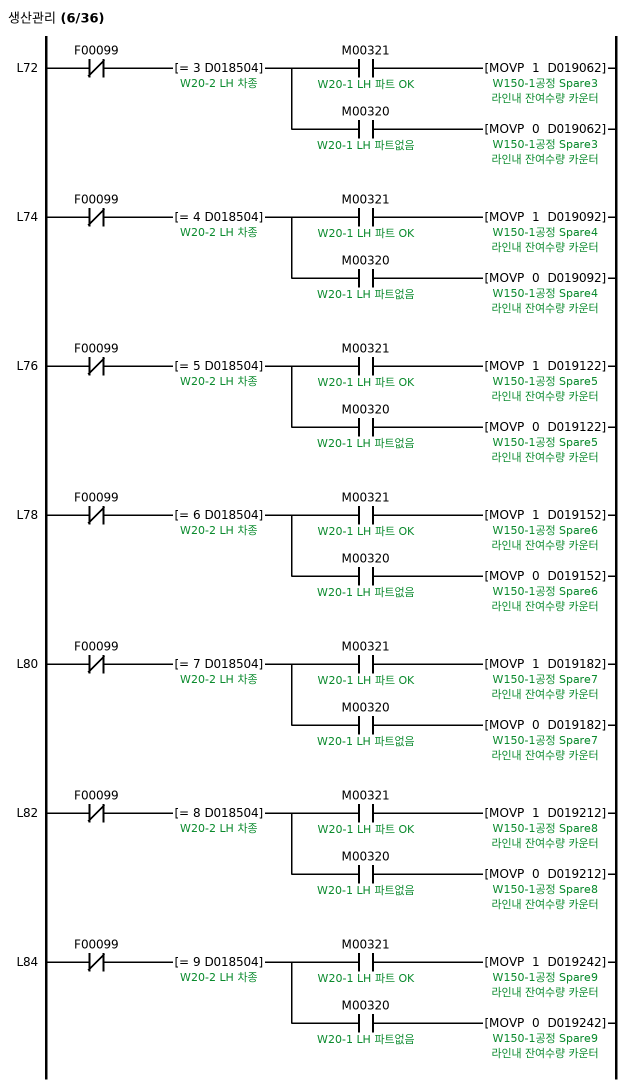
; L72
LOAD NOT  F00099
AND=      3 D018504	// W20-2 LH 차종
MPUSH
AND       M00321	// W20-1 LH 파트 OK
MOVP      1 D019062	// W150-1공정 Spare3 라인내 잔여수량 카운터
MPOP
AND       M00320	// W20-1 LH 파트없음
MOVP      0 D019062	// W150-1공정 Spare3 라인내 잔여수량 카운터
; L74
LOAD NOT  F00099
AND=      4 D018504	// W20-2 LH 차종
MPUSH
AND       M00321	// W20-1 LH 파트 OK
MOVP      1 D019092	// W150-1공정 Spare4 라인내 잔여수량 카운터
MPOP
AND       M00320	// W20-1 LH 파트없음
MOVP      0 D019092	// W150-1공정 Spare4 라인내 잔여수량 카운터
; L76
LOAD NOT  F00099
AND=      5 D018504	// W20-2 LH 차종
MPUSH
AND       M00321	// W20-1 LH 파트 OK
MOVP      1 D019122	// W150-1공정 Spare5 라인내 잔여수량 카운터
MPOP
AND       M00320	// W20-1 LH 파트없음
MOVP      0 D019122	// W150-1공정 Spare5 라인내 잔여수량 카운터
; L78
LOAD NOT  F00099
AND=      6 D018504	// W20-2 LH 차종
MPUSH
AND       M00321	// W20-1 LH 파트 OK
MOVP      1 D019152	// W150-1공정 Spare6 라인내 잔여수량 카운터
MPOP
AND       M00320	// W20-1 LH 파트없음
MOVP      0 D019152	// W150-1공정 Spare6 라인내 잔여수량 카운터
; L80
LOAD NOT  F00099
AND=      7 D018504	// W20-2 LH 차종
MPUSH
AND       M00321	// W20-1 LH 파트 OK
MOVP      1 D019182	// W150-1공정 Spare7 라인내 잔여수량 카운터
MPOP
AND       M00320	// W20-1 LH 파트없음
MOVP      0 D019182	// W150-1공정 Spare7 라인내 잔여수량 카운터
; L82
LOAD NOT  F00099
AND=      8 D018504	// W20-2 LH 차종
MPUSH
AND       M00321	// W20-1 LH 파트 OK
MOVP      1 D019212	// W150-1공정 Spare8 라인내 잔여수량 카운터
MPOP
AND       M00320	// W20-1 LH 파트없음
MOVP      0 D019212	// W150-1공정 Spare8 라인내 잔여수량 카운터
; L84
LOAD NOT  F00099
AND=      9 D018504	// W20-2 LH 차종
MPUSH
AND       M00321	// W20-1 LH 파트 OK
MOVP      1 D019242	// W150-1공정 Spare9 라인내 잔여수량 카운터
MPOP
AND       M00320	// W20-1 LH 파트없음
MOVP      0 D019242	// W150-1공정 Spare9 라인내 잔여수량 카운터

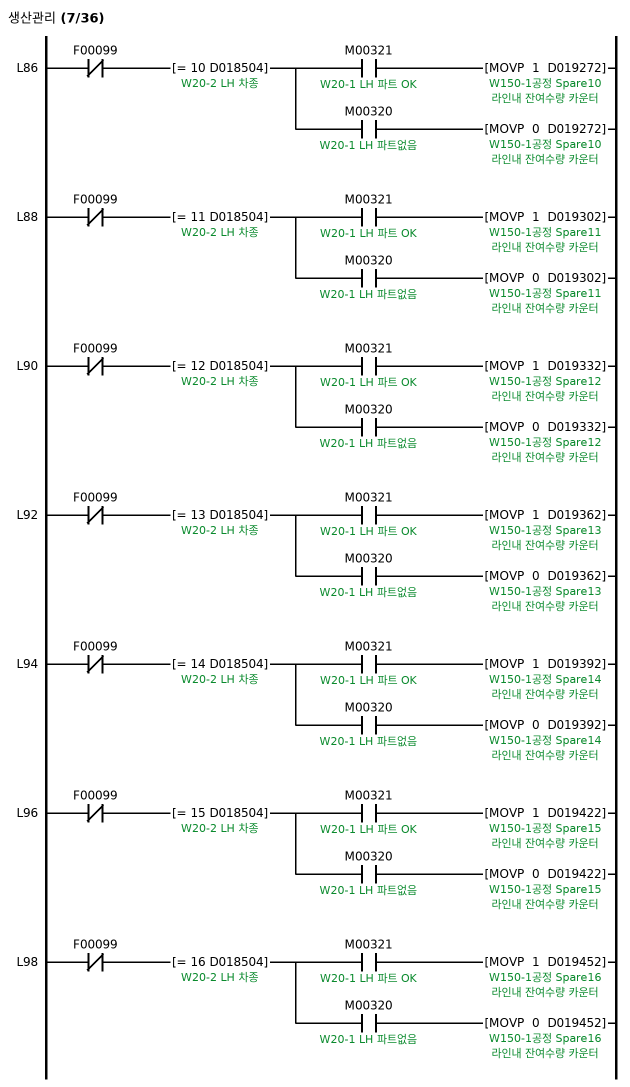
; L86
LOAD NOT  F00099
AND=      10 D018504	// W20-2 LH 차종
MPUSH
AND       M00321	// W20-1 LH 파트 OK
MOVP      1 D019272	// W150-1공정 Spare10 라인내 잔여수량 카운터
MPOP
AND       M00320	// W20-1 LH 파트없음
MOVP      0 D019272	// W150-1공정 Spare10 라인내 잔여수량 카운터
; L88
LOAD NOT  F00099
AND=      11 D018504	// W20-2 LH 차종
MPUSH
AND       M00321	// W20-1 LH 파트 OK
MOVP      1 D019302	// W150-1공정 Spare11 라인내 잔여수량 카운터
MPOP
AND       M00320	// W20-1 LH 파트없음
MOVP      0 D019302	// W150-1공정 Spare11 라인내 잔여수량 카운터
; L90
LOAD NOT  F00099
AND=      12 D018504	// W20-2 LH 차종
MPUSH
AND       M00321	// W20-1 LH 파트 OK
MOVP      1 D019332	// W150-1공정 Spare12 라인내 잔여수량 카운터
MPOP
AND       M00320	// W20-1 LH 파트없음
MOVP      0 D019332	// W150-1공정 Spare12 라인내 잔여수량 카운터
; L92
LOAD NOT  F00099
AND=      13 D018504	// W20-2 LH 차종
MPUSH
AND       M00321	// W20-1 LH 파트 OK
MOVP      1 D019362	// W150-1공정 Spare13 라인내 잔여수량 카운터
MPOP
AND       M00320	// W20-1 LH 파트없음
MOVP      0 D019362	// W150-1공정 Spare13 라인내 잔여수량 카운터
; L94
LOAD NOT  F00099
AND=      14 D018504	// W20-2 LH 차종
MPUSH
AND       M00321	// W20-1 LH 파트 OK
MOVP      1 D019392	// W150-1공정 Spare14 라인내 잔여수량 카운터
MPOP
AND       M00320	// W20-1 LH 파트없음
MOVP      0 D019392	// W150-1공정 Spare14 라인내 잔여수량 카운터
; L96
LOAD NOT  F00099
AND=      15 D018504	// W20-2 LH 차종
MPUSH
AND       M00321	// W20-1 LH 파트 OK
MOVP      1 D019422	// W150-1공정 Spare15 라인내 잔여수량 카운터
MPOP
AND       M00320	// W20-1 LH 파트없음
MOVP      0 D019422	// W150-1공정 Spare15 라인내 잔여수량 카운터
; L98
LOAD NOT  F00099
AND=      16 D018504	// W20-2 LH 차종
MPUSH
AND       M00321	// W20-1 LH 파트 OK
MOVP      1 D019452	// W150-1공정 Spare16 라인내 잔여수량 카운터
MPOP
AND       M00320	// W20-1 LH 파트없음
MOVP      0 D019452	// W150-1공정 Spare16 라인내 잔여수량 카운터

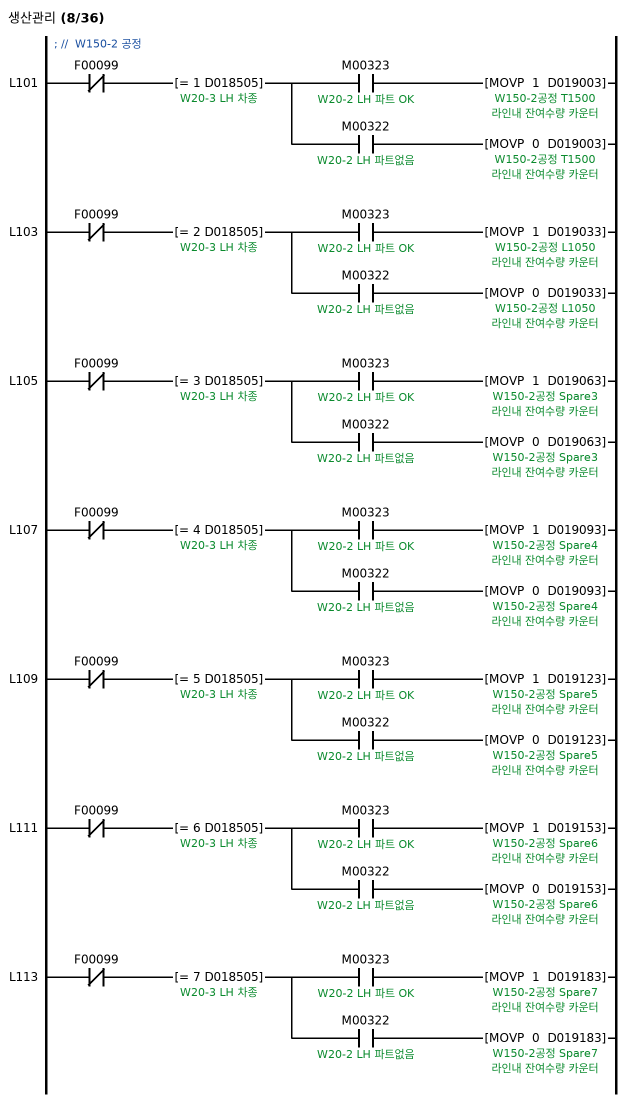
//   //  W150-2 공정
; L101
LOAD NOT  F00099
AND=      1 D018505	// W20-3 LH 차종
MPUSH
AND       M00323	// W20-2 LH 파트 OK
MOVP      1 D019003	// W150-2공정 T1500 라인내 잔여수량 카운터
MPOP
AND       M00322	// W20-2 LH 파트없음
MOVP      0 D019003	// W150-2공정 T1500 라인내 잔여수량 카운터
; L103
LOAD NOT  F00099
AND=      2 D018505	// W20-3 LH 차종
MPUSH
AND       M00323	// W20-2 LH 파트 OK
MOVP      1 D019033	// W150-2공정 L1050 라인내 잔여수량 카운터
MPOP
AND       M00322	// W20-2 LH 파트없음
MOVP      0 D019033	// W150-2공정 L1050 라인내 잔여수량 카운터
; L105
LOAD NOT  F00099
AND=      3 D018505	// W20-3 LH 차종
MPUSH
AND       M00323	// W20-2 LH 파트 OK
MOVP      1 D019063	// W150-2공정 Spare3 라인내 잔여수량 카운터
MPOP
AND       M00322	// W20-2 LH 파트없음
MOVP      0 D019063	// W150-2공정 Spare3 라인내 잔여수량 카운터
; L107
LOAD NOT  F00099
AND=      4 D018505	// W20-3 LH 차종
MPUSH
AND       M00323	// W20-2 LH 파트 OK
MOVP      1 D019093	// W150-2공정 Spare4 라인내 잔여수량 카운터
MPOP
AND       M00322	// W20-2 LH 파트없음
MOVP      0 D019093	// W150-2공정 Spare4 라인내 잔여수량 카운터
; L109
LOAD NOT  F00099
AND=      5 D018505	// W20-3 LH 차종
MPUSH
AND       M00323	// W20-2 LH 파트 OK
MOVP      1 D019123	// W150-2공정 Spare5 라인내 잔여수량 카운터
MPOP
AND       M00322	// W20-2 LH 파트없음
MOVP      0 D019123	// W150-2공정 Spare5 라인내 잔여수량 카운터
; L111
LOAD NOT  F00099
AND=      6 D018505	// W20-3 LH 차종
MPUSH
AND       M00323	// W20-2 LH 파트 OK
MOVP      1 D019153	// W150-2공정 Spare6 라인내 잔여수량 카운터
MPOP
AND       M00322	// W20-2 LH 파트없음
MOVP      0 D019153	// W150-2공정 Spare6 라인내 잔여수량 카운터
; L113
LOAD NOT  F00099
AND=      7 D018505	// W20-3 LH 차종
MPUSH
AND       M00323	// W20-2 LH 파트 OK
MOVP      1 D019183	// W150-2공정 Spare7 라인내 잔여수량 카운터
MPOP
AND       M00322	// W20-2 LH 파트없음
MOVP      0 D019183	// W150-2공정 Spare7 라인내 잔여수량 카운터

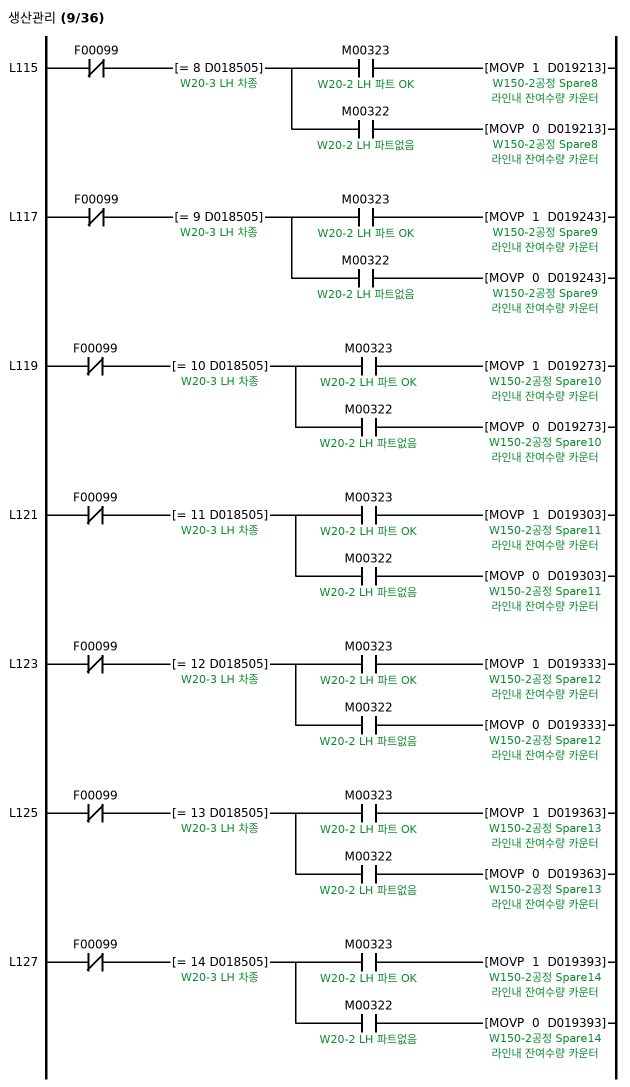
; L115
LOAD NOT  F00099
AND=      8 D018505	// W20-3 LH 차종
MPUSH
AND       M00323	// W20-2 LH 파트 OK
MOVP      1 D019213	// W150-2공정 Spare8 라인내 잔여수량 카운터
MPOP
AND       M00322	// W20-2 LH 파트없음
MOVP      0 D019213	// W150-2공정 Spare8 라인내 잔여수량 카운터
; L117
LOAD NOT  F00099
AND=      9 D018505	// W20-3 LH 차종
MPUSH
AND       M00323	// W20-2 LH 파트 OK
MOVP      1 D019243	// W150-2공정 Spare9 라인내 잔여수량 카운터
MPOP
AND       M00322	// W20-2 LH 파트없음
MOVP      0 D019243	// W150-2공정 Spare9 라인내 잔여수량 카운터
; L119
LOAD NOT  F00099
AND=      10 D018505	// W20-3 LH 차종
MPUSH
AND       M00323	// W20-2 LH 파트 OK
MOVP      1 D019273	// W150-2공정 Spare10 라인내 잔여수량 카운터
MPOP
AND       M00322	// W20-2 LH 파트없음
MOVP      0 D019273	// W150-2공정 Spare10 라인내 잔여수량 카운터
; L121
LOAD NOT  F00099
AND=      11 D018505	// W20-3 LH 차종
MPUSH
AND       M00323	// W20-2 LH 파트 OK
MOVP      1 D019303	// W150-2공정 Spare11 라인내 잔여수량 카운터
MPOP
AND       M00322	// W20-2 LH 파트없음
MOVP      0 D019303	// W150-2공정 Spare11 라인내 잔여수량 카운터
; L123
LOAD NOT  F00099
AND=      12 D018505	// W20-3 LH 차종
MPUSH
AND       M00323	// W20-2 LH 파트 OK
MOVP      1 D019333	// W150-2공정 Spare12 라인내 잔여수량 카운터
MPOP
AND       M00322	// W20-2 LH 파트없음
MOVP      0 D019333	// W150-2공정 Spare12 라인내 잔여수량 카운터
; L125
LOAD NOT  F00099
AND=      13 D018505	// W20-3 LH 차종
MPUSH
AND       M00323	// W20-2 LH 파트 OK
MOVP      1 D019363	// W150-2공정 Spare13 라인내 잔여수량 카운터
MPOP
AND       M00322	// W20-2 LH 파트없음
MOVP      0 D019363	// W150-2공정 Spare13 라인내 잔여수량 카운터
; L127
LOAD NOT  F00099
AND=      14 D018505	// W20-3 LH 차종
MPUSH
AND       M00323	// W20-2 LH 파트 OK
MOVP      1 D019393	// W150-2공정 Spare14 라인내 잔여수량 카운터
MPOP
AND       M00322	// W20-2 LH 파트없음
MOVP      0 D019393	// W150-2공정 Spare14 라인내 잔여수량 카운터

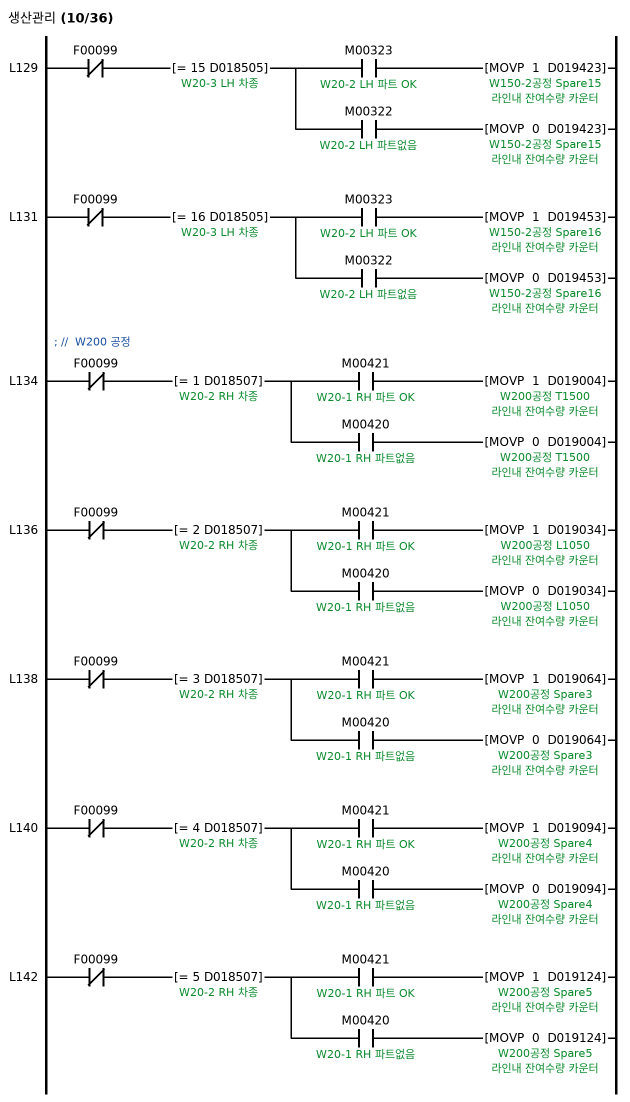
; L129
LOAD NOT  F00099
AND=      15 D018505	// W20-3 LH 차종
MPUSH
AND       M00323	// W20-2 LH 파트 OK
MOVP      1 D019423	// W150-2공정 Spare15 라인내 잔여수량 카운터
MPOP
AND       M00322	// W20-2 LH 파트없음
MOVP      0 D019423	// W150-2공정 Spare15 라인내 잔여수량 카운터
; L131
LOAD NOT  F00099
AND=      16 D018505	// W20-3 LH 차종
MPUSH
AND       M00323	// W20-2 LH 파트 OK
MOVP      1 D019453	// W150-2공정 Spare16 라인내 잔여수량 카운터
MPOP
AND       M00322	// W20-2 LH 파트없음
MOVP      0 D019453	// W150-2공정 Spare16 라인내 잔여수량 카운터
//   //  W200 공정
; L134
LOAD NOT  F00099
AND=      1 D018507	// W20-2 RH 차종
MPUSH
AND       M00421	// W20-1 RH 파트 OK
MOVP      1 D019004	// W200공정 T1500 라인내 잔여수량 카운터
MPOP
AND       M00420	// W20-1 RH 파트없음
MOVP      0 D019004	// W200공정 T1500 라인내 잔여수량 카운터
; L136
LOAD NOT  F00099
AND=      2 D018507	// W20-2 RH 차종
MPUSH
AND       M00421	// W20-1 RH 파트 OK
MOVP      1 D019034	// W200공정 L1050 라인내 잔여수량 카운터
MPOP
AND       M00420	// W20-1 RH 파트없음
MOVP      0 D019034	// W200공정 L1050 라인내 잔여수량 카운터
; L138
LOAD NOT  F00099
AND=      3 D018507	// W20-2 RH 차종
MPUSH
AND       M00421	// W20-1 RH 파트 OK
MOVP      1 D019064	// W200공정 Spare3 라인내 잔여수량 카운터
MPOP
AND       M00420	// W20-1 RH 파트없음
MOVP      0 D019064	// W200공정 Spare3 라인내 잔여수량 카운터
; L140
LOAD NOT  F00099
AND=      4 D018507	// W20-2 RH 차종
MPUSH
AND       M00421	// W20-1 RH 파트 OK
MOVP      1 D019094	// W200공정 Spare4 라인내 잔여수량 카운터
MPOP
AND       M00420	// W20-1 RH 파트없음
MOVP      0 D019094	// W200공정 Spare4 라인내 잔여수량 카운터
; L142
LOAD NOT  F00099
AND=      5 D018507	// W20-2 RH 차종
MPUSH
AND       M00421	// W20-1 RH 파트 OK
MOVP      1 D019124	// W200공정 Spare5 라인내 잔여수량 카운터
MPOP
AND       M00420	// W20-1 RH 파트없음
MOVP      0 D019124	// W200공정 Spare5 라인내 잔여수량 카운터

